LIN {X 0,Y 368.171,Z 278.475,A -85,B 0,C 180,E1 12084.523,E2 12084.523} C_VEL
LIN {X 0,Y 365.845,Z 275.09,A -85,B 0,C 180,E1 12082.497,E2 12082.497} C_VEL
LIN {X 0,Y 364.939,Z 273.089,A -85,B 0,C 180,E1 12081.371,E2 12081.371} C_VEL
LIN {X 0,Y 362.071,Z 268.956,A -85,B 0,C 180,E1 12077.685,E2 12077.685} C_VEL
LIN {X 0,Y 361.817,Z 267.734,A -85,B 0,C 180,E1 12076.208,E2 12076.208} C_VEL
LIN {X 0,Y 361.806,Z 267.661,A -85,B 0,C 180,E1 12072.125,E2 12072.125} C_VEL
LIN {X 0,Y 361.806,Z 267.652,A -85,B 0,C 180,E1 12067.943,E2 12067.943} C_VEL
LIN {X 0,Y 361.86,Z 268.035,A -85,B 0,C 180,E1 12064.438,E2 12064.438} C_VEL
LIN {X 0,Y 364.418,Z 272.635,A -85,B 0,C 180,E1 12060.316,E2 12060.316} C_VEL
LIN {X 0,Y 365.404,Z 274.131,A -85,B 0,C 180,E1 12059.217,E2 12059.217} C_VEL
LIN {X 0,Y 367.498,Z 277.914,A -85,B 0,C 180,E1 12057.038,E2 12057.038} C_VEL
LIN {X 0,Y 368.456,Z 279.19,A -85,B 0,C 180,E1 12056.267,E2 12056.267} C_VEL
LIN {X 0,Y 370.329,Z 282.88,A -85,B 0,C 180,E1 12054.579,E2 12054.579} C_VEL
LIN {X 0,Y 371.35,Z 284.531,A -85,B 0,C 180,E1 12053.819,E2 12053.819} C_VEL
LIN {X 0,Y 373.993,Z 289.456,A -85,B 0,C 180,E1 12051.856,E2 12051.856} C_VEL
LIN {X 0,Y 376.746,Z 294.987,A -85,B 0,C 180,E1 12049.913,E2 12049.913} C_VEL
LIN {X 0,Y 379.817,Z 300.91,A -85,B 0,C 180,E1 12048.075,E2 12048.075} C_VEL
LIN {X 0,Y 385.945,Z 309.361,A -85,B 0,C 180,E1 12046.293,E2 12046.293} C_VEL
LIN {X 0,Y 394.032,Z 321.193,A -85,B 0,C 180,E1 12044.158,E2 12044.158} C_VEL
LIN {X 0,Y 402.897,Z 335.236,A -85,B 0,C 180,E1 12042.042,E2 12042.042} C_VEL
LIN {X 0,Y 410.49,Z 348.634,A -85,B 0,C 180,E1 12040.362,E2 12040.362} C_VEL
LIN {X 0,Y 399.537,Z 571.468,A -85,B 0,C 180,E1 12035.877,E2 12035.877} C_VEL
LIN {X 0,Y 397.756,Z 592.269,A -85,B 0,C 180,E1 12035.206,E2 12035.206} C_VEL
LIN {X 0,Y 395.491,Z 611.619,A -85,B 0,C 180,E1 12034.346,E2 12034.346} C_VEL
LIN {X 0,Y 392.522,Z 632.048,A -85,B 0,C 180,E1 12033.159,E2 12033.159} C_VEL
LIN {X 0,Y 389.245,Z 650.935,A -85,B 0,C 180,E1 12031.774,E2 12031.774} C_VEL
LIN {X 0,Y 385.65,Z 668.995,A -85,B 0,C 180,E1 12030.148,E2 12030.148} C_VEL
LIN {X 0,Y 381.789,Z 686.588,A -85,B 0,C 180,E1 12028.209,E2 12028.209} C_VEL
LIN {X 0,Y 377.954,Z 702.615,A -85,B 0,C 180,E1 12026.071,E2 12026.071} C_VEL
LIN {X 0,Y 374.362,Z 717.031,A -85,B 0,C 180,E1 12023.766,E2 12023.766} C_VEL
LIN {X 0,Y 370.819,Z 731.031,A -85,B 0,C 180,E1 12021.081,E2 12021.081} C_VEL
LIN {X 0,Y 367.884,Z 742.762,A -85,B 0,C 180,E1 12018.369,E2 12018.369} C_VEL
LIN {X 0,Y 365.466,Z 752.896,A -85,B 0,C 180,E1 12015.546,E2 12015.546} C_VEL
LIN {X 0,Y 363.43,Z 762.078,A -85,B 0,C 180,E1 12012.381,E2 12012.381} C_VEL
LIN {X 0,Y 362.031,Z 769.268,A -85,B 0,C 180,E1 12009.233,E2 12009.233} C_VEL
LIN {X 0,Y 361.116,Z 774.969,A -85,B 0,C 180,E1 12005.945,E2 12005.945} C_VEL
LIN {X 0,Y 360.61,Z 779.064,A -85,B 0,C 180,E1 12002.542,E2 12002.542} C_VEL
LIN {X 0,Y 360.405,Z 781.321,A -85,B 0,C 180,E1 11999.411,E2 11999.411} C_VEL
LIN {X 0,Y 360.342,Z 782.079,A -85,B 0,C 180,E1 11996.336,E2 11996.336} C_VEL
LIN {X 0,Y 360.361,Z 781.41,A -85,B 0,C 180,E1 11993.205,E2 11993.205} C_VEL
LIN {X 0,Y 360.519,Z 779.191,A -85,B 0,C 180,E1 11989.925,E2 11989.925} C_VEL
LIN {X 0,Y 360.9,Z 775.517,A -85,B 0,C 180,E1 11986.747,E2 11986.747} C_VEL
LIN {X 0,Y 361.665,Z 769.902,A -85,B 0,C 180,E1 11983.43,E2 11983.43} C_VEL
LIN {X 0,Y 362.853,Z 762.904,A -85,B 0,C 180,E1 11980.32,E2 11980.32} C_VEL
LIN {X 0,Y 364.579,Z 754.204,A -85,B 0,C 180,E1 11977.249,E2 11977.249} C_VEL
LIN {X 0,Y 366.111,Z 747.184,A -85,B 0,C 180,E1 11975.17,E2 11975.17} C_VEL
LIN {X 0,Y 366.048,Z 743.524,A -85,B 0,C 180,E1 11974.098,E2 11974.098} C_VEL
LIN {X 0,Y 362.759,Z 733.509,A -85,B 0,C 180,E1 11971.203,E2 11971.203} C_VEL
LIN {X 0,Y 363.017,Z 729.697,A -85,B 0,C 180,E1 11970.335,E2 11970.335} C_VEL
LIN {X 0,Y 366.543,Z 715.603,A -85,B 0,C 180,E1 11967.657,E2 11967.657} C_VEL
LIN {X 0,Y 370.168,Z 700.835,A -85,B 0,C 180,E1 11965.319,E2 11965.319} C_VEL
LIN {X 0,Y 373.855,Z 685.185,A -85,B 0,C 180,E1 11963.244,E2 11963.244} C_VEL
LIN {X 0,Y 377.797,Z 666.968,A -85,B 0,C 180,E1 11961.249,E2 11961.249} C_VEL
LIN {X 0,Y 381.444,Z 648.231,A -85,B 0,C 180,E1 11959.582,E2 11959.582} C_VEL
LIN {X 0,Y 384.61,Z 629.426,A -85,B 0,C 180,E1 11958.226,E2 11958.226} C_VEL
LIN {X 0,Y 387.367,Z 609.919,A -85,B 0,C 180,E1 11957.108,E2 11957.108} C_VEL
LIN {X 0,Y 389.704,Z 589.326,A -85,B 0,C 180,E1 11956.212,E2 11956.212} C_VEL
LIN {X 0,Y 391.382,Z 568.754,A -85,B 0,C 180,E1 11955.569,E2 11955.569} C_VEL
LIN {X 0,Y 401.198,Z 349.516,A -85,B 0,C 180,E1 11951.239,E2 11951.239} C_VEL
LIN {X 0,Y 390.797,Z 331.837,A -85,B 0,C 180,E1 11949.151,E2 11949.151} C_VEL
LIN {X 0,Y 380.876,Z 316.345,A -85,B 0,C 180,E1 11947.024,E2 11947.024} C_VEL
LIN {X 0,Y 369.459,Z 299.547,A -85,B 0,C 180,E1 11944.31,E2 11944.31} C_VEL
LIN {X 0,Y 363.406,Z 287.193,A -85,B 0,C 180,E1 11941.032,E2 11941.032} C_VEL
LIN {X 0,Y 360.31,Z 281.531,A -85,B 0,C 180,E1 11939.34,E2 11939.34} C_VEL
LIN {X 0,Y 358.366,Z 277.681,A -85,B 0,C 180,E1 11938.178,E2 11938.178} C_VEL
LIN {X 0,Y 356.111,Z 273.295,A -85,B 0,C 180,E1 11936.789,E2 11936.789} C_VEL
LIN {X 0,Y 354.135,Z 269.94,A -85,B 0,C 180,E1 11935.623,E2 11935.623} C_VEL
LIN {X 0,Y 353.858,Z 268.676,A -85,B 0,C 180,E1 11935.1,E2 11935.1} C_VEL
LIN {X 0,Y 353.852,Z 268.637,A -85,B 0,C 180,E1 11930.944,E2 11930.944} C_VEL
LIN {X 0,Y 353.853,Z 268.639,A -85,B 0,C 180,E1 11926.801,E2 11926.801} C_VEL
LIN {X 0,Y 353.855,Z 268.648,A -85,B 0,C 180,E1 11922.696,E2 11922.696} C_VEL
LIN {X 0,Y 353.858,Z 268.656,A -85,B 0,C 180,E1 11918.433,E2 11918.433} C_VEL
LIN {X 0,Y 353.864,Z 268.647,A -85,B 0,C 180,E1 11914.122,E2 11914.122} C_VEL
LIN {X 0,Y 353.873,Z 268.628,A -85,B 0,C 180,E1 11909.818,E2 11909.818} C_VEL
LIN {X 0,Y 353.866,Z 268.625,A -85,B 0,C 180,E1 11905.612,E2 11905.612} C_VEL
LIN {X 0,Y 353.872,Z 268.643,A -85,B 0,C 180,E1 11901.374,E2 11901.374} C_VEL
LIN {X 0,Y 353.864,Z 268.654,A -85,B 0,C 180,E1 11897.087,E2 11897.087} C_VEL
LIN {X 0,Y 353.859,Z 268.629,A -85,B 0,C 180,E1 11892.894,E2 11892.894} C_VEL
LIN {X 0,Y 353.856,Z 268.625,A -85,B 0,C 180,E1 11888.775,E2 11888.775} C_VEL
LIN {X 0,Y 353.857,Z 268.649,A -85,B 0,C 180,E1 11884.699,E2 11884.699} C_VEL
LIN {X 0,Y 353.854,Z 268.656,A -85,B 0,C 180,E1 11880.484,E2 11880.484} C_VEL
LIN {X 0,Y 353.847,Z 268.636,A -85,B 0,C 180,E1 11876.272,E2 11876.272} C_VEL
LIN {X 0,Y 353.843,Z 268.629,A -85,B 0,C 180,E1 11872.04,E2 11872.04} C_VEL
LIN {X 0,Y 353.844,Z 268.63,A -85,B 0,C 180,E1 11867.864,E2 11867.864} C_VEL
LIN {X 0,Y 353.844,Z 268.637,A -85,B 0,C 180,E1 11863.754,E2 11863.754} C_VEL
LIN {X 0,Y 353.846,Z 268.64,A -85,B 0,C 180,E1 11859.661,E2 11859.661} C_VEL
LIN {X 0,Y 353.913,Z 268.942,A -85,B 0,C 180,E1 11856.655,E2 11856.655} C_VEL
LIN {X 0,Y 355.339,Z 272.39,A -85,B 0,C 180,E1 11855.566,E2 11855.566} C_VEL
LIN {X 0,Y 356.893,Z 274.427,A -85,B 0,C 180,E1 11854.795,E2 11854.795} C_VEL
LIN {X 0,Y 358.766,Z 278.091,A -85,B 0,C 180,E1 11853.696,E2 11853.696} C_VEL
LIN {X 0,Y 359.707,Z 279.455,A -85,B 0,C 180,E1 11853.236,E2 11853.236} C_VEL
LIN {X 0,Y 362.062,Z 283.638,A -85,B 0,C 180,E1 11851.999,E2 11851.999} C_VEL
LIN {X 0,Y 368.063,Z 295.125,A -85,B 0,C 180,E1 11848.925,E2 11848.925} C_VEL
LIN {X 0,Y 371.968,Z 302.135,A -85,B 0,C 180,E1 11847.227,E2 11847.227} C_VEL
LIN {X 0,Y 385.1,Z 320.964,A -85,B 0,C 180,E1 11844.208,E2 11844.208} C_VEL
LIN {X 0,Y 397.504,Z 340.13,A -85,B 0,C 180,E1 11841.612,E2 11841.612} C_VEL
LIN {X 0,Y 405.844,Z 354.423,A -85,B 0,C 180,E1 11839.974,E2 11839.974} C_VEL
LIN {X 0,Y 397.273,Z 565.921,A -85,B 0,C 180,E1 11835.942,E2 11835.942} C_VEL
LIN {X 0,Y 395.586,Z 604.161,A -85,B 0,C 180,E1 11835.173,E2 11835.173} C_VEL
LIN {X 0,Y 393.543,Z 625.831,A -85,B 0,C 180,E1 11834.533,E2 11834.533} C_VEL
LIN {X 0,Y 390.884,Z 646.572,A -85,B 0,C 180,E1 11833.678,E2 11833.678} C_VEL
LIN {X 0,Y 387.766,Z 666.981,A -85,B 0,C 180,E1 11832.585,E2 11832.585} C_VEL
LIN {X 0,Y 384.063,Z 687.555,A -85,B 0,C 180,E1 11831.195,E2 11831.195} C_VEL
LIN {X 0,Y 380.11,Z 706.817,A -85,B 0,C 180,E1 11829.581,E2 11829.581} C_VEL
LIN {X 0,Y 375.81,Z 726.104,A -85,B 0,C 180,E1 11827.63,E2 11827.63} C_VEL
LIN {X 0,Y 371.717,Z 743.57,A -85,B 0,C 180,E1 11825.519,E2 11825.519} C_VEL
LIN {X 0,Y 367.661,Z 760.077,A -85,B 0,C 180,E1 11823.133,E2 11823.133} C_VEL
LIN {X 0,Y 363.946,Z 775.21,A -85,B 0,C 180,E1 11820.545,E2 11820.545} C_VEL
LIN {X 0,Y 360.639,Z 789.096,A -85,B 0,C 180,E1 11817.758,E2 11817.758} C_VEL
LIN {X 0,Y 357.812,Z 801.747,A -85,B 0,C 180,E1 11814.745,E2 11814.745} C_VEL
LIN {X 0,Y 355.593,Z 812.75,A -85,B 0,C 180,E1 11811.612,E2 11811.612} C_VEL
LIN {X 0,Y 353.937,Z 822.534,A -85,B 0,C 180,E1 11808.273,E2 11808.273} C_VEL
LIN {X 0,Y 352.897,Z 830.469,A -85,B 0,C 180,E1 11804.939,E2 11804.939} C_VEL
LIN {X 0,Y 352.357,Z 836.632,A -85,B 0,C 180,E1 11801.621,E2 11801.621} C_VEL
LIN {X 0,Y 352.155,Z 841.286,A -85,B 0,C 180,E1 11798.324,E2 11798.324} C_VEL
LIN {X 0,Y 352.148,Z 844.279,A -85,B 0,C 180,E1 11795.048,E2 11795.048} C_VEL
LIN {X 0,Y 352.177,Z 845.844,A -85,B 0,C 180,E1 11791.788,E2 11791.788} C_VEL
LIN {X 0,Y 352.189,Z 845.904,A -85,B 0,C 180,E1 11788.86,E2 11788.86} C_VEL
LIN {X 0,Y 352.155,Z 844.641,A -85,B 0,C 180,E1 11785.602,E2 11785.602} C_VEL
LIN {X 0,Y 352.151,Z 841.936,A -85,B 0,C 180,E1 11782.494,E2 11782.494} C_VEL
LIN {X 0,Y 352.305,Z 837.422,A -85,B 0,C 180,E1 11779.037,E2 11779.037} C_VEL
LIN {X 0,Y 352.749,Z 831.577,A -85,B 0,C 180,E1 11775.789,E2 11775.789} C_VEL
LIN {X 0,Y 353.717,Z 823.505,A -85,B 0,C 180,E1 11772.291,E2 11772.291} C_VEL
LIN {X 0,Y 355.282,Z 813.801,A -85,B 0,C 180,E1 11768.884,E2 11768.884} C_VEL
LIN {X 0,Y 357.524,Z 802.262,A -85,B 0,C 180,E1 11765.548,E2 11765.548} C_VEL
LIN {X 0,Y 360.232,Z 789.837,A -85,B 0,C 180,E1 11762.563,E2 11762.563} C_VEL
LIN {X 0,Y 363.661,Z 775.346,A -85,B 0,C 180,E1 11759.608,E2 11759.608} C_VEL
LIN {X 0,Y 367.455,Z 759.895,A -85,B 0,C 180,E1 11756.939,E2 11756.939} C_VEL
LIN {X 0,Y 371.492,Z 743.408,A -85,B 0,C 180,E1 11754.547,E2 11754.547} C_VEL
LIN {X 0,Y 375.747,Z 725.523,A -85,B 0,C 180,E1 11752.359,E2 11752.359} C_VEL
LIN {X 0,Y 380.019,Z 706.741,A -85,B 0,C 180,E1 11750.436,E2 11750.436} C_VEL
LIN {X 0,Y 384.069,Z 687.407,A -85,B 0,C 180,E1 11748.796,E2 11748.796} C_VEL
LIN {X 0,Y 387.78,Z 667.348,A -85,B 0,C 180,E1 11747.42,E2 11747.42} C_VEL
LIN {X 0,Y 391.268,Z 645.478,A -85,B 0,C 180,E1 11746.229,E2 11746.229} C_VEL
LIN {X 0,Y 394.075,Z 624.25,A -85,B 0,C 180,E1 11745.354,E2 11745.354} C_VEL
LIN {X 0,Y 396.163,Z 602.513,A -85,B 0,C 180,E1 11744.713,E2 11744.713} C_VEL
LIN {X 0,Y 397.935,Z 563.509,A -85,B 0,C 180,E1 11743.924,E2 11743.924} C_VEL
LIN {X 0,Y 406.612,Z 362.247,A -85,B 0,C 180,E1 11740.032,E2 11740.032} C_VEL
LIN {X 0,Y 406.892,Z 353.823,A -85,B 0,C 180,E1 11739.848,E2 11739.848} C_VEL
LIN {X 0,Y 398.203,Z 338.538,A -85,B 0,C 180,E1 11737.897,E2 11737.897} C_VEL
LIN {X 0,Y 389.857,Z 325.331,A -85,B 0,C 180,E1 11735.86,E2 11735.86} C_VEL
LIN {X 0,Y 381.451,Z 313.134,A -85,B 0,C 180,E1 11733.579,E2 11733.579} C_VEL
LIN {X 0,Y 374.48,Z 303.819,A -85,B 0,C 180,E1 11731.466,E2 11731.466} C_VEL
LIN {X 0,Y 372.423,Z 300.702,A -85,B 0,C 180,E1 11730.671,E2 11730.671} C_VEL
LIN {X 0,Y 369.278,Z 294.916,A -85,B 0,C 180,E1 11728.637,E2 11728.637} C_VEL
LIN {X 0,Y 366.686,Z 290.179,A -85,B 0,C 180,E1 11726.739,E2 11726.739} C_VEL
LIN {X 0,Y 364.476,Z 286.447,A -85,B 0,C 180,E1 11724.991,E2 11724.991} C_VEL
LIN {X 0,Y 363.776,Z 285.103,A -85,B 0,C 180,E1 11724.349,E2 11724.349} C_VEL
LIN {X 0,Y 361.487,Z 281.641,A -85,B 0,C 180,E1 11722.269,E2 11722.269} C_VEL
LIN {X 0,Y 360.76,Z 279.896,A -85,B 0,C 180,E1 11721.29,E2 11721.29} C_VEL
LIN {X 0,Y 357.919,Z 275.754,A -85,B 0,C 180,E1 11717.561,E2 11717.561} C_VEL
LIN {X 0,Y 357.203,Z 274.236,A -85,B 0,C 180,E1 11715.922,E2 11715.922} C_VEL
LIN {X 0,Y 355.791,Z 272.948,A -85,B 0,C 180,E1 11711.182,E2 11711.182} C_VEL
LIN {X 0,Y 356.483,Z 273.641,A -85,B 0,C 180,E1 11706.825,E2 11706.825} C_VEL
LIN {X 0,Y 357.675,Z 274.972,A -85,B 0,C 180,E1 11704.33,E2 11704.33} C_VEL
LIN {X 0,Y 360.059,Z 279.305,A -85,B 0,C 180,E1 11700.479,E2 11700.479} C_VEL
LIN {X 0,Y 360.971,Z 280.593,A -85,B 0,C 180,E1 11699.471,E2 11699.471} C_VEL
LIN {X 0,Y 363.034,Z 284.512,A -85,B 0,C 180,E1 11697.16,E2 11697.16} C_VEL
LIN {X 0,Y 363.802,Z 285.478,A -85,B 0,C 180,E1 11696.535,E2 11696.535} C_VEL
LIN {X 0,Y 365.818,Z 289.463,A -85,B 0,C 180,E1 11694.669,E2 11694.669} C_VEL
LIN {X 0,Y 366.727,Z 291.216,A -85,B 0,C 180,E1 11693.898,E2 11693.898} C_VEL
LIN {X 0,Y 369.138,Z 295.706,A -85,B 0,C 180,E1 11692.061,E2 11692.061} C_VEL
LIN {X 0,Y 371.718,Z 300.754,A -85,B 0,C 180,E1 11690.284,E2 11690.284} C_VEL
LIN {X 0,Y 379.116,Z 310.838,A -85,B 0,C 180,E1 11687.86,E2 11687.86} C_VEL
LIN {X 0,Y 384.806,Z 318.805,A -85,B 0,C 180,E1 11686.209,E2 11686.209} C_VEL
LIN {X 0,Y 393.452,Z 331.999,A -85,B 0,C 180,E1 11683.921,E2 11683.921} C_VEL
LIN {X 0,Y 402.593,Z 347.489,A -85,B 0,C 180,E1 11681.728,E2 11681.728} C_VEL
LIN {X 0,Y 405.119,Z 352.351,A -85,B 0,C 180,E1 11681.15,E2 11681.15} C_VEL
LIN {X 0,Y 393.789,Z 571.901,A -85,B 0,C 180,E1 11676.678,E2 11676.678} C_VEL
LIN {X 0,Y 391.933,Z 592.665,A -85,B 0,C 180,E1 11676.003,E2 11676.003} C_VEL
LIN {X 0,Y 389.485,Z 612.63,A -85,B 0,C 180,E1 11675.103,E2 11675.103} C_VEL
LIN {X 0,Y 386.367,Z 633.083,A -85,B 0,C 180,E1 11673.896,E2 11673.896} C_VEL
LIN {X 0,Y 382.894,Z 652.166,A -85,B 0,C 180,E1 11672.472,E2 11672.472} C_VEL
LIN {X 0,Y 379.319,Z 669.352,A -85,B 0,C 180,E1 11670.906,E2 11670.906} C_VEL
LIN {X 0,Y 375.234,Z 687.046,A -85,B 0,C 180,E1 11668.933,E2 11668.933} C_VEL
LIN {X 0,Y 371.199,Z 703.146,A -85,B 0,C 180,E1 11666.76,E2 11666.76} C_VEL
LIN {X 0,Y 367.346,Z 717.828,A -85,B 0,C 180,E1 11664.378,E2 11664.378} C_VEL
LIN {X 0,Y 363.718,Z 731.354,A -85,B 0,C 180,E1 11661.743,E2 11661.743} C_VEL
LIN {X 0,Y 360.512,Z 743.426,A -85,B 0,C 180,E1 11658.908,E2 11658.908} C_VEL
LIN {X 0,Y 357.828,Z 753.961,A -85,B 0,C 180,E1 11655.901,E2 11655.901} C_VEL
LIN {X 0,Y 355.665,Z 763.142,A -85,B 0,C 180,E1 11652.651,E2 11652.651} C_VEL
LIN {X 0,Y 354.14,Z 770.471,A -85,B 0,C 180,E1 11649.325,E2 11649.325} C_VEL
LIN {X 0,Y 353.201,Z 775.872,A -85,B 0,C 180,E1 11646.075,E2 11646.075} C_VEL
LIN {X 0,Y 352.66,Z 779.898,A -85,B 0,C 180,E1 11642.596,E2 11642.596} C_VEL
LIN {X 0,Y 352.43,Z 782.154,A -85,B 0,C 180,E1 11639.209,E2 11639.209} C_VEL
LIN {X 0,Y 352.37,Z 782.827,A -85,B 0,C 180,E1 11635.913,E2 11635.913} C_VEL
LIN {X 0,Y 352.41,Z 781.93,A -85,B 0,C 180,E1 11632.699,E2 11632.699} C_VEL
LIN {X 0,Y 352.604,Z 779.492,A -85,B 0,C 180,E1 11629.378,E2 11629.378} C_VEL
LIN {X 0,Y 353.091,Z 775.301,A -85,B 0,C 180,E1 11625.944,E2 11625.944} C_VEL
LIN {X 0,Y 353.951,Z 769.762,A -85,B 0,C 180,E1 11622.73,E2 11622.73} C_VEL
LIN {X 0,Y 355.386,Z 762.171,A -85,B 0,C 180,E1 11619.393,E2 11619.393} C_VEL
LIN {X 0,Y 357.464,Z 752.599,A -85,B 0,C 180,E1 11616.103,E2 11616.103} C_VEL
LIN {X 0,Y 359.942,Z 742.108,A -85,B 0,C 180,E1 11613.186,E2 11613.186} C_VEL
LIN {X 0,Y 362.943,Z 729.991,A -85,B 0,C 180,E1 11610.397,E2 11610.397} C_VEL
LIN {X 0,Y 363.017,Z 729.697,A -85,B 0,C 180,E1 11610.335,E2 11610.335} C_VEL
LIN {X 0,Y 363.276,Z 725.23,A -85,B 0,C 180,E1 11609.334,E2 11609.334} C_VEL
LIN {X 0,Y 360.943,Z 713.902,A -85,B 0,C 180,E1 11606.727,E2 11606.727} C_VEL
LIN {X 0,Y 361.384,Z 708.797,A -85,B 0,C 180,E1 11605.802,E2 11605.802} C_VEL
LIN {X 0,Y 365.243,Z 693.476,A -85,B 0,C 180,E1 11603.554,E2 11603.554} C_VEL
LIN {X 0,Y 369.208,Z 676.766,A -85,B 0,C 180,E1 11601.514,E2 11601.514} C_VEL
LIN {X 0,Y 373.175,Z 658.233,A -85,B 0,C 180,E1 11599.66,E2 11599.66} C_VEL
LIN {X 0,Y 376.74,Z 639.384,A -85,B 0,C 180,E1 11598.132,E2 11598.132} C_VEL
LIN {X 0,Y 379.858,Z 620.033,A -85,B 0,C 180,E1 11596.874,E2 11596.874} C_VEL
LIN {X 0,Y 382.617,Z 598.881,A -85,B 0,C 180,E1 11595.808,E2 11595.808} C_VEL
LIN {X 0,Y 384.726,Z 577.543,A -85,B 0,C 180,E1 11595.029,E2 11595.029} C_VEL
LIN {X 0,Y 386.119,Z 555.392,A -85,B 0,C 180,E1 11594.487,E2 11594.487} C_VEL
LIN {X 0,Y 395.493,Z 352.855,A -85,B 0,C 180,E1 11590.469,E2 11590.469} C_VEL
LIN {X 0,Y 384.578,Z 334.275,A -85,B 0,C 180,E1 11588.194,E2 11588.194} C_VEL
LIN {X 0,Y 373.601,Z 317.34,A -85,B 0,C 180,E1 11585.723,E2 11585.723} C_VEL
LIN {X 0,Y 364.389,Z 304.199,A -85,B 0,C 180,E1 11583.486,E2 11583.486} C_VEL
LIN {X 0,Y 361.111,Z 299.359,A -85,B 0,C 180,E1 11582.55,E2 11582.55} C_VEL
LIN {X 0,Y 355.957,Z 288.76,A -85,B 0,C 180,E1 11579.576,E2 11579.576} C_VEL
LIN {X 0,Y 352.905,Z 283.238,A -85,B 0,C 180,E1 11577.818,E2 11577.818} C_VEL
LIN {X 0,Y 350.988,Z 279.336,A -85,B 0,C 180,E1 11576.577,E2 11576.577} C_VEL
LIN {X 0,Y 348.936,Z 275.745,A -85,B 0,C 180,E1 11575.32,E2 11575.32} C_VEL
LIN {X 0,Y 348.005,Z 274.092,A -85,B 0,C 180,E1 11574.728,E2 11574.728} C_VEL
LIN {X 0,Y 346.094,Z 270.562,A -85,B 0,C 180,E1 11573.427,E2 11573.427} C_VEL
LIN {X 0,Y 345.919,Z 269.661,A -85,B 0,C 180,E1 11572.838,E2 11572.838} C_VEL
LIN {X 0,Y 345.922,Z 269.637,A -85,B 0,C 180,E1 11568.558,E2 11568.558} C_VEL
LIN {X 0,Y 345.926,Z 269.633,A -85,B 0,C 180,E1 11564.211,E2 11564.211} C_VEL
LIN {X 0,Y 345.931,Z 269.621,A -85,B 0,C 180,E1 11559.913,E2 11559.913} C_VEL
LIN {X 0,Y 345.925,Z 269.613,A -85,B 0,C 180,E1 11555.692,E2 11555.692} C_VEL
LIN {X 0,Y 345.931,Z 269.615,A -85,B 0,C 180,E1 11551.503,E2 11551.503} C_VEL
LIN {X 0,Y 345.928,Z 269.637,A -85,B 0,C 180,E1 11547.171,E2 11547.171} C_VEL
LIN {X 0,Y 345.923,Z 269.641,A -85,B 0,C 180,E1 11542.965,E2 11542.965} C_VEL
LIN {X 0,Y 345.913,Z 269.616,A -85,B 0,C 180,E1 11538.712,E2 11538.712} C_VEL
LIN {X 0,Y 345.908,Z 269.612,A -85,B 0,C 180,E1 11534.468,E2 11534.468} C_VEL
LIN {X 0,Y 345.911,Z 269.634,A -85,B 0,C 180,E1 11530.154,E2 11530.154} C_VEL
LIN {X 0,Y 345.914,Z 269.647,A -85,B 0,C 180,E1 11525.971,E2 11525.971} C_VEL
LIN {X 0,Y 345.919,Z 269.622,A -85,B 0,C 180,E1 11521.655,E2 11521.655} C_VEL
LIN {X 0,Y 345.918,Z 269.613,A -85,B 0,C 180,E1 11517.514,E2 11517.514} C_VEL
LIN {X 0,Y 345.935,Z 269.616,A -85,B 0,C 180,E1 11513.193,E2 11513.193} C_VEL
LIN {X 0,Y 345.928,Z 269.628,A -85,B 0,C 180,E1 11509.001,E2 11509.001} C_VEL
LIN {X 0,Y 345.933,Z 269.637,A -85,B 0,C 180,E1 11504.75,E2 11504.75} C_VEL
LIN {X 0,Y 345.919,Z 269.638,A -85,B 0,C 180,E1 11500.409,E2 11500.409} C_VEL
LIN {X 0,Y 345.974,Z 269.9,A -85,B 0,C 180,E1 11498.822,E2 11498.822} C_VEL
LIN {X 0,Y 347.342,Z 273.305,A -85,B 0,C 180,E1 11497.667,E2 11497.667} C_VEL
LIN {X 0,Y 348.915,Z 275.084,A -85,B 0,C 180,E1 11496.883,E2 11496.883} C_VEL
LIN {X 0,Y 350.583,Z 278.721,A -85,B 0,C 180,E1 11495.751,E2 11495.751} C_VEL
LIN {X 0,Y 351.847,Z 280.308,A -85,B 0,C 180,E1 11495.128,E2 11495.128} C_VEL
LIN {X 0,Y 354.001,Z 284.439,A -85,B 0,C 180,E1 11493.856,E2 11493.856} C_VEL
LIN {X 0,Y 357.753,Z 291.307,A -85,B 0,C 180,E1 11491.814,E2 11491.814} C_VEL
LIN {X 0,Y 362.576,Z 300.412,A -85,B 0,C 180,E1 11489.324,E2 11489.324} C_VEL
LIN {X 0,Y 365.385,Z 304.531,A -85,B 0,C 180,E1 11488.488,E2 11488.488} C_VEL
LIN {X 0,Y 376.936,Z 320.677,A -85,B 0,C 180,E1 11485.689,E2 11485.689} C_VEL
LIN {X 0,Y 388.911,Z 339.001,A -85,B 0,C 180,E1 11483.038,E2 11483.038} C_VEL
LIN {X 0,Y 399.643,Z 356.661,A -85,B 0,C 180,E1 11480.845,E2 11480.845} C_VEL
LIN {X 0,Y 400.16,Z 358.051,A -85,B 0,C 180,E1 11480.73,E2 11480.73} C_VEL
LIN {X 0,Y 391.142,Z 571.042,A -85,B 0,C 180,E1 11476.627,E2 11476.627} C_VEL
LIN {X 0,Y 389.53,Z 604.571,A -85,B 0,C 180,E1 11475.933,E2 11475.933} C_VEL
LIN {X 0,Y 387.377,Z 626.504,A -85,B 0,C 180,E1 11475.275,E2 11475.275} C_VEL
LIN {X 0,Y 384.526,Z 647.648,A -85,B 0,C 180,E1 11474.381,E2 11474.381} C_VEL
LIN {X 0,Y 381.112,Z 668.76,A -85,B 0,C 180,E1 11473.212,E2 11473.212} C_VEL
LIN {X 0,Y 377.47,Z 688.165,A -85,B 0,C 180,E1 11471.872,E2 11471.872} C_VEL
LIN {X 0,Y 373.282,Z 707.629,A -85,B 0,C 180,E1 11470.203,E2 11470.203} C_VEL
LIN {X 0,Y 368.898,Z 726.345,A -85,B 0,C 180,E1 11468.264,E2 11468.264} C_VEL
LIN {X 0,Y 364.484,Z 744.244,A -85,B 0,C 180,E1 11466.042,E2 11466.042} C_VEL
LIN {X 0,Y 360.335,Z 760.447,A -85,B 0,C 180,E1 11463.649,E2 11463.649} C_VEL
LIN {X 0,Y 356.526,Z 775.178,A -85,B 0,C 180,E1 11461.063,E2 11461.063} C_VEL
LIN {X 0,Y 352.879,Z 789.692,A -85,B 0,C 180,E1 11458.055,E2 11458.055} C_VEL
LIN {X 0,Y 349.983,Z 802.091,A -85,B 0,C 180,E1 11455.01,E2 11455.01} C_VEL
LIN {X 0,Y 347.625,Z 813.216,A -85,B 0,C 180,E1 11451.714,E2 11451.714} C_VEL
LIN {X 0,Y 345.888,Z 823.044,A -85,B 0,C 180,E1 11448.19,E2 11448.19} C_VEL
LIN {X 0,Y 344.858,Z 830.757,A -85,B 0,C 180,E1 11444.78,E2 11444.78} C_VEL
LIN {X 0,Y 344.338,Z 836.699,A -85,B 0,C 180,E1 11441.386,E2 11441.386} C_VEL
LIN {X 0,Y 344.164,Z 841.257,A -85,B 0,C 180,E1 11437.831,E2 11437.831} C_VEL
LIN {X 0,Y 344.172,Z 843.917,A -85,B 0,C 180,E1 11434.664,E2 11434.664} C_VEL
LIN {X 0,Y 344.214,Z 845.199,A -85,B 0,C 180,E1 11431.33,E2 11431.33} C_VEL
LIN {X 0,Y 344.214,Z 845.106,A -85,B 0,C 180,E1 11428.334,E2 11428.334} C_VEL
LIN {X 0,Y 344.182,Z 843.549,A -85,B 0,C 180,E1 11424.999,E2 11424.999} C_VEL
LIN {X 0,Y 344.183,Z 840.681,A -85,B 0,C 180,E1 11421.815,E2 11421.815} C_VEL
LIN {X 0,Y 344.385,Z 835.855,A -85,B 0,C 180,E1 11418.272,E2 11418.272} C_VEL
LIN {X 0,Y 344.942,Z 829.639,A -85,B 0,C 180,E1 11414.851,E2 11414.851} C_VEL
LIN {X 0,Y 346.043,Z 821.52,A -85,B 0,C 180,E1 11411.394,E2 11411.394} C_VEL
LIN {X 0,Y 347.844,Z 811.38,A -85,B 0,C 180,E1 11407.878,E2 11407.878} C_VEL
LIN {X 0,Y 350.227,Z 800.163,A -85,B 0,C 180,E1 11404.643,E2 11404.643} C_VEL
LIN {X 0,Y 353.38,Z 786.828,A -85,B 0,C 180,E1 11401.432,E2 11401.432} C_VEL
LIN {X 0,Y 356.9,Z 772.756,A -85,B 0,C 180,E1 11398.594,E2 11398.594} C_VEL
LIN {X 0,Y 361.285,Z 755.881,A -85,B 0,C 180,E1 11395.722,E2 11395.722} C_VEL
LIN {X 0,Y 365.487,Z 739.624,A -85,B 0,C 180,E1 11393.387,E2 11393.387} C_VEL
LIN {X 0,Y 369.956,Z 721.639,A -85,B 0,C 180,E1 11391.23,E2 11391.23} C_VEL
LIN {X 0,Y 374.398,Z 702.656,A -85,B 0,C 180,E1 11389.335,E2 11389.335} C_VEL
LIN {X 0,Y 378.729,Z 682.354,A -85,B 0,C 180,E1 11387.665,E2 11387.665} C_VEL
LIN {X 0,Y 382.633,Z 661.929,A -85,B 0,C 180,E1 11386.312,E2 11386.312} C_VEL
LIN {X 0,Y 385.824,Z 641.882,A -85,B 0,C 180,E1 11385.272,E2 11385.272} C_VEL
LIN {X 0,Y 388.686,Z 620.024,A -85,B 0,C 180,E1 11384.412,E2 11384.412} C_VEL
LIN {X 0,Y 390.704,Z 598.338,A -85,B 0,C 180,E1 11383.799,E2 11383.799} C_VEL
LIN {X 0,Y 400.982,Z 371.603,A -85,B 0,C 180,E1 11379.349,E2 11379.349} C_VEL
LIN {X 0,Y 401.57,Z 357.268,A -85,B 0,C 180,E1 11379.046,E2 11379.046} C_VEL
LIN {X 0,Y 393.149,Z 342.514,A -85,B 0,C 180,E1 11377.067,E2 11377.067} C_VEL
LIN {X 0,Y 384.57,Z 328.75,A -85,B 0,C 180,E1 11374.844,E2 11374.844} C_VEL
LIN {X 0,Y 376.015,Z 316.302,A -85,B 0,C 180,E1 11372.354,E2 11372.354} C_VEL
LIN {X 0,Y 368.313,Z 306.134,A -85,B 0,C 180,E1 11369.789,E2 11369.789} C_VEL
LIN {X 0,Y 364.545,Z 301.13,A -85,B 0,C 180,E1 11368.328,E2 11368.328} C_VEL
LIN {X 0,Y 361.97,Z 296.448,A -85,B 0,C 180,E1 11366.407,E2 11366.407} C_VEL
LIN {X 0,Y 359.79,Z 292.186,A -85,B 0,C 180,E1 11364.462,E2 11364.462} C_VEL
LIN {X 0,Y 357.159,Z 288.205,A -85,B 0,C 180,E1 11362.033,E2 11362.033} C_VEL
LIN {X 0,Y 356.409,Z 286.551,A -85,B 0,C 180,E1 11361.045,E2 11361.045} C_VEL
LIN {X 0,Y 353.667,Z 282.15,A -85,B 0,C 180,E1 11357.1,E2 11357.1} C_VEL
LIN {X 0,Y 352.939,Z 280.965,A -85,B 0,C 180,E1 11355.445,E2 11355.445} C_VEL
LIN {X 0,Y 351.763,Z 279.859,A -85,B 0,C 180,E1 11351.146,E2 11351.146} C_VEL
LIN {X 0,Y 352.407,Z 280.524,A -85,B 0,C 180,E1 11346.845,E2 11346.845} C_VEL
LIN {X 0,Y 353.511,Z 281.84,A -85,B 0,C 180,E1 11344.381,E2 11344.381} C_VEL
LIN {X 0,Y 355.843,Z 286.109,A -85,B 0,C 180,E1 11340.484,E2 11340.484} C_VEL
LIN {X 0,Y 356.617,Z 287.448,A -85,B 0,C 180,E1 11339.519,E2 11339.519} C_VEL
LIN {X 0,Y 358.785,Z 291.326,A -85,B 0,C 180,E1 11337.126,E2 11337.126} C_VEL
LIN {X 0,Y 359.644,Z 293.306,A -85,B 0,C 180,E1 11336.164,E2 11336.164} C_VEL
LIN {X 0,Y 361.856,Z 297.08,A -85,B 0,C 180,E1 11334.293,E2 11334.293} C_VEL
LIN {X 0,Y 364.193,Z 301.205,A -85,B 0,C 180,E1 11332.588,E2 11332.588} C_VEL
LIN {X 0,Y 371.844,Z 311.501,A -85,B 0,C 180,E1 11329.752,E2 11329.752} C_VEL
LIN {X 0,Y 379.217,Z 321.892,A -85,B 0,C 180,E1 11327.403,E2 11327.403} C_VEL
LIN {X 0,Y 387.109,Z 333.881,A -85,B 0,C 180,E1 11325.167,E2 11325.167} C_VEL
LIN {X 0,Y 395.407,Z 347.595,A -85,B 0,C 180,E1 11323.039,E2 11323.039} C_VEL
LIN {X 0,Y 399.855,Z 355.851,A -85,B 0,C 180,E1 11321.964,E2 11321.964} C_VEL
LIN {X 0,Y 388.118,Z 572.484,A -85,B 0,C 180,E1 11317.501,E2 11317.501} C_VEL
LIN {X 0,Y 386.187,Z 593.234,A -85,B 0,C 180,E1 11316.819,E2 11316.819} C_VEL
LIN {X 0,Y 383.641,Z 613.206,A -85,B 0,C 180,E1 11315.911,E2 11315.911} C_VEL
LIN {X 0,Y 380.424,Z 633.425,A -85,B 0,C 180,E1 11314.708,E2 11314.708} C_VEL
LIN {X 0,Y 376.869,Z 652.182,A -85,B 0,C 180,E1 11313.3,E2 11313.3} C_VEL
LIN {X 0,Y 372.843,Z 670.616,A -85,B 0,C 180,E1 11311.596,E2 11311.596} C_VEL
LIN {X 0,Y 368.611,Z 688.152,A -85,B 0,C 180,E1 11309.609,E2 11309.609} C_VEL
LIN {X 0,Y 364.373,Z 704.205,A -85,B 0,C 180,E1 11307.399,E2 11307.399} C_VEL
LIN {X 0,Y 360.442,Z 718.377,A -85,B 0,C 180,E1 11305.058,E2 11305.058} C_VEL
LIN {X 0,Y 356.477,Z 732.395,A -85,B 0,C 180,E1 11302.277,E2 11302.277} C_VEL
LIN {X 0,Y 353.061,Z 744.514,A -85,B 0,C 180,E1 11299.359,E2 11299.359} C_VEL
LIN {X 0,Y 350.233,Z 754.931,A -85,B 0,C 180,E1 11296.304,E2 11296.304} C_VEL
LIN {X 0,Y 348.027,Z 763.683,A -85,B 0,C 180,E1 11293.14,E2 11293.14} C_VEL
LIN {X 0,Y 346.406,Z 770.837,A -85,B 0,C 180,E1 11289.849,E2 11289.849} C_VEL
LIN {X 0,Y 345.381,Z 776.211,A -85,B 0,C 180,E1 11286.611,E2 11286.611} C_VEL
LIN {X 0,Y 344.781,Z 780.216,A -85,B 0,C 180,E1 11283.238,E2 11283.238} C_VEL
LIN {X 0,Y 344.503,Z 782.7,A -85,B 0,C 180,E1 11279.801,E2 11279.801} C_VEL
LIN {X 0,Y 344.406,Z 783.5,A -85,B 0,C 180,E1 11276.558,E2 11276.558} C_VEL
LIN {X 0,Y 344.426,Z 782.903,A -85,B 0,C 180,E1 11273.255,E2 11273.255} C_VEL
LIN {X 0,Y 344.597,Z 780.864,A -85,B 0,C 180,E1 11269.939,E2 11269.939} C_VEL
LIN {X 0,Y 345.04,Z 777.128,A -85,B 0,C 180,E1 11266.5,E2 11266.5} C_VEL
LIN {X 0,Y 345.896,Z 771.639,A -85,B 0,C 180,E1 11263.067,E2 11263.067} C_VEL
LIN {X 0,Y 347.247,Z 764.666,A -85,B 0,C 180,E1 11259.783,E2 11259.783} C_VEL
LIN {X 0,Y 349.302,Z 755.552,A -85,B 0,C 180,E1 11256.411,E2 11256.411} C_VEL
LIN {X 0,Y 351.934,Z 744.943,A -85,B 0,C 180,E1 11253.259,E2 11253.259} C_VEL
LIN {X 0,Y 354.946,Z 733.428,A -85,B 0,C 180,E1 11250.441,E2 11250.441} C_VEL
LIN {X 0,Y 358.428,Z 720.249,A -85,B 0,C 180,E1 11247.764,E2 11247.764} C_VEL
LIN {X 0,Y 361.384,Z 708.797,A -85,B 0,C 180,E1 11245.802,E2 11245.802} C_VEL
LIN {X 0,Y 361.903,Z 703.596,A -85,B 0,C 180,E1 11244.891,E2 11244.891} C_VEL
LIN {X 0,Y 360.223,Z 690.498,A -85,B 0,C 180,E1 11242.481,E2 11242.481} C_VEL
LIN {X 0,Y 360.8,Z 684.716,A -85,B 0,C 180,E1 11241.666,E2 11241.666} C_VEL
LIN {X 0,Y 364.877,Z 667.388,A -85,B 0,C 180,E1 11239.742,E2 11239.742} C_VEL
LIN {X 0,Y 368.842,Z 648.511,A -85,B 0,C 180,E1 11238.033,E2 11238.033} C_VEL
LIN {X 0,Y 372.277,Z 629.481,A -85,B 0,C 180,E1 11236.647,E2 11236.647} C_VEL
LIN {X 0,Y 375.289,Z 609.52,A -85,B 0,C 180,E1 11235.498,E2 11235.498} C_VEL
LIN {X 0,Y 377.815,Z 588.282,A -85,B 0,C 180,E1 11234.578,E2 11234.578} C_VEL
LIN {X 0,Y 379.558,Z 567.452,A -85,B 0,C 180,E1 11233.94,E2 11233.94} C_VEL
LIN {X 0,Y 389.827,Z 356.154,A -85,B 0,C 180,E1 11229.677,E2 11229.677} C_VEL
LIN {X 0,Y 378.988,Z 337.794,A -85,B 0,C 180,E1 11227.332,E2 11227.332} C_VEL
LIN {X 0,Y 368.203,Z 321.085,A -85,B 0,C 180,E1 11224.811,E2 11224.811} C_VEL
LIN {X 0,Y 358.535,Z 307.221,A -85,B 0,C 180,E1 11222.342,E2 11222.342} C_VEL
LIN {X 0,Y 353.197,Z 299.841,A -85,B 0,C 180,E1 11220.865,E2 11220.865} C_VEL
LIN {X 0,Y 348.271,Z 289.95,A -85,B 0,C 180,E1 11217.874,E2 11217.874} C_VEL
LIN {X 0,Y 345.481,Z 284.886,A -85,B 0,C 180,E1 11216.157,E2 11216.157} C_VEL
LIN {X 0,Y 343.062,Z 280.304,A -85,B 0,C 180,E1 11214.553,E2 11214.553} C_VEL
LIN {X 0,Y 341.04,Z 276.601,A -85,B 0,C 180,E1 11213.163,E2 11213.163} C_VEL
LIN {X 0,Y 338.287,Z 272.026,A -85,B 0,C 180,E1 11211.284,E2 11211.284} C_VEL
LIN {X 0,Y 337.984,Z 270.653,A -85,B 0,C 180,E1 11210.65,E2 11210.65} C_VEL
LIN {X 0,Y 337.982,Z 270.609,A -85,B 0,C 180,E1 11206.429,E2 11206.429} C_VEL
LIN {X 0,Y 337.989,Z 270.61,A -85,B 0,C 180,E1 11202.057,E2 11202.057} C_VEL
LIN {X 0,Y 337.993,Z 270.62,A -85,B 0,C 180,E1 11197.757,E2 11197.757} C_VEL
LIN {X 0,Y 337.991,Z 270.633,A -85,B 0,C 180,E1 11193.381,E2 11193.381} C_VEL
LIN {X 0,Y 337.984,Z 270.618,A -85,B 0,C 180,E1 11189.021,E2 11189.021} C_VEL
LIN {X 0,Y 337.973,Z 270.603,A -85,B 0,C 180,E1 11184.744,E2 11184.744} C_VEL
LIN {X 0,Y 337.971,Z 270.605,A -85,B 0,C 180,E1 11180.43,E2 11180.43} C_VEL
LIN {X 0,Y 337.975,Z 270.628,A -85,B 0,C 180,E1 11176.144,E2 11176.144} C_VEL
LIN {X 0,Y 337.976,Z 270.624,A -85,B 0,C 180,E1 11171.95,E2 11171.95} C_VEL
LIN {X 0,Y 337.987,Z 270.602,A -85,B 0,C 180,E1 11167.649,E2 11167.649} C_VEL
LIN {X 0,Y 337.984,Z 270.603,A -85,B 0,C 180,E1 11163.39,E2 11163.39} C_VEL
LIN {X 0,Y 337.994,Z 270.617,A -85,B 0,C 180,E1 11159.151,E2 11159.151} C_VEL
LIN {X 0,Y 337.985,Z 270.632,A -85,B 0,C 180,E1 11154.737,E2 11154.737} C_VEL
LIN {X 0,Y 337.982,Z 270.622,A -85,B 0,C 180,E1 11150.635,E2 11150.635} C_VEL
LIN {X 0,Y 337.973,Z 270.616,A -85,B 0,C 180,E1 11146.309,E2 11146.309} C_VEL
LIN {X 0,Y 337.969,Z 270.615,A -85,B 0,C 180,E1 11142.08,E2 11142.08} C_VEL
LIN {X 0,Y 338.043,Z 271.002,A -85,B 0,C 180,E1 11141.165,E2 11141.165} C_VEL
LIN {X 0,Y 339.577,Z 274.524,A -85,B 0,C 180,E1 11139.848,E2 11139.848} C_VEL
LIN {X 0,Y 341.079,Z 276.1,A -85,B 0,C 180,E1 11139.044,E2 11139.044} C_VEL
LIN {X 0,Y 342.9,Z 280.008,A -85,B 0,C 180,E1 11137.723,E2 11137.723} C_VEL
LIN {X 0,Y 344.086,Z 281.546,A -85,B 0,C 180,E1 11137.083,E2 11137.083} C_VEL
LIN {X 0,Y 346.126,Z 285.438,A -85,B 0,C 180,E1 11135.782,E2 11135.782} C_VEL
LIN {X 0,Y 347.217,Z 287.377,A -85,B 0,C 180,E1 11135.137,E2 11135.137} C_VEL
LIN {X 0,Y 349.999,Z 292.433,A -85,B 0,C 180,E1 11133.534,E2 11133.534} C_VEL
LIN {X 0,Y 354.742,Z 301.048,A -85,B 0,C 180,E1 11131,E2 11131} C_VEL
LIN {X 0,Y 366.044,Z 316.682,A -85,B 0,C 180,E1 11127.953,E2 11127.953} C_VEL
LIN {X 0,Y 377.169,Z 332.913,A -85,B 0,C 180,E1 11125.275,E2 11125.275} C_VEL
LIN {X 0,Y 389.332,Z 352.124,A -85,B 0,C 180,E1 11122.6,E2 11122.6} C_VEL
LIN {X 0,Y 394.531,Z 361.269,A -85,B 0,C 180,E1 11121.511,E2 11121.511} C_VEL
LIN {X 0,Y 385.058,Z 576.371,A -85,B 0,C 180,E1 11117.33,E2 11117.33} C_VEL
LIN {X 0,Y 383.447,Z 606.098,A -85,B 0,C 180,E1 11116.688,E2 11116.688} C_VEL
LIN {X 0,Y 381.176,Z 627.82,A -85,B 0,C 180,E1 11116.014,E2 11116.014} C_VEL
LIN {X 0,Y 378.197,Z 648.865,A -85,B 0,C 180,E1 11115.098,E2 11115.098} C_VEL
LIN {X 0,Y 374.691,Z 669.424,A -85,B 0,C 180,E1 11113.929,E2 11113.929} C_VEL
LIN {X 0,Y 370.713,Z 689.517,A -85,B 0,C 180,E1 11112.5,E2 11112.5} C_VEL
LIN {X 0,Y 366.397,Z 708.825,A -85,B 0,C 180,E1 11110.809,E2 11110.809} C_VEL
LIN {X 0,Y 361.86,Z 727.266,A -85,B 0,C 180,E1 11108.843,E2 11108.843} C_VEL
LIN {X 0,Y 357.208,Z 745.189,A -85,B 0,C 180,E1 11106.549,E2 11106.549} C_VEL
LIN {X 0,Y 352.809,Z 761.586,A -85,B 0,C 180,E1 11104.05,E2 11104.05} C_VEL
LIN {X 0,Y 348.675,Z 776.863,A -85,B 0,C 180,E1 11101.265,E2 11101.265} C_VEL
LIN {X 0,Y 345.127,Z 790.275,A -85,B 0,C 180,E1 11098.365,E2 11098.365} C_VEL
LIN {X 0,Y 342.129,Z 802.469,A -85,B 0,C 180,E1 11095.255,E2 11095.255} C_VEL
LIN {X 0,Y 339.627,Z 813.826,A -85,B 0,C 180,E1 11091.772,E2 11091.772} C_VEL
LIN {X 0,Y 337.907,Z 823.113,A -85,B 0,C 180,E1 11088.277,E2 11088.277} C_VEL
LIN {X 0,Y 336.816,Z 831.011,A -85,B 0,C 180,E1 11084.588,E2 11084.588} C_VEL
LIN {X 0,Y 336.322,Z 836.763,A -85,B 0,C 180,E1 11081.14,E2 11081.14} C_VEL
LIN {X 0,Y 336.179,Z 840.855,A -85,B 0,C 180,E1 11077.69,E2 11077.69} C_VEL
LIN {X 0,Y 336.201,Z 843.516,A -85,B 0,C 180,E1 11074.262,E2 11074.262} C_VEL
LIN {X 0,Y 336.25,Z 844.529,A -85,B 0,C 180,E1 11071.02,E2 11071.02} C_VEL
LIN {X 0,Y 336.236,Z 844.257,A -85,B 0,C 180,E1 11067.659,E2 11067.659} C_VEL
LIN {X 0,Y 336.197,Z 842.449,A -85,B 0,C 180,E1 11064.366,E2 11064.366} C_VEL
LIN {X 0,Y 336.215,Z 839.116,A -85,B 0,C 180,E1 11060.87,E2 11060.87} C_VEL
LIN {X 0,Y 336.481,Z 834.289,A -85,B 0,C 180,E1 11057.47,E2 11057.47} C_VEL
LIN {X 0,Y 337.207,Z 827.43,A -85,B 0,C 180,E1 11053.814,E2 11053.814} C_VEL
LIN {X 0,Y 338.489,Z 819.188,A -85,B 0,C 180,E1 11050.32,E2 11050.32} C_VEL
LIN {X 0,Y 340.516,Z 808.853,A -85,B 0,C 180,E1 11046.791,E2 11046.791} C_VEL
LIN {X 0,Y 343.268,Z 796.929,A -85,B 0,C 180,E1 11043.409,E2 11043.409} C_VEL
LIN {X 0,Y 346.678,Z 783.606,A -85,B 0,C 180,E1 11040.242,E2 11040.242} C_VEL
LIN {X 0,Y 350.737,Z 768.612,A -85,B 0,C 180,E1 11037.243,E2 11037.243} C_VEL
LIN {X 0,Y 355.122,Z 752.437,A -85,B 0,C 180,E1 11034.548,E2 11034.548} C_VEL
LIN {X 0,Y 359.843,Z 734.967,A -85,B 0,C 180,E1 11032.104,E2 11032.104} C_VEL
LIN {X 0,Y 364.56,Z 716.684,A -85,B 0,C 180,E1 11029.961,E2 11029.961} C_VEL
LIN {X 0,Y 369.165,Z 697.655,A -85,B 0,C 180,E1 11028.114,E2 11028.114} C_VEL
LIN {X 0,Y 373.312,Z 678.581,A -85,B 0,C 180,E1 11026.606,E2 11026.606} C_VEL
LIN {X 0,Y 377.445,Z 657.052,A -85,B 0,C 180,E1 11025.231,E2 11025.231} C_VEL
LIN {X 0,Y 380.631,Z 637.629,A -85,B 0,C 180,E1 11024.252,E2 11024.252} C_VEL
LIN {X 0,Y 383.398,Z 616,A -85,B 0,C 180,E1 11023.446,E2 11023.446} C_VEL
LIN {X 0,Y 385.335,Z 593.528,A -85,B 0,C 180,E1 11022.852,E2 11022.852} C_VEL
LIN {X 0,Y 395.792,Z 373.825,A -85,B 0,C 180,E1 11018.499,E2 11018.499} C_VEL
LIN {X 0,Y 396.36,Z 360.835,A -85,B 0,C 180,E1 11018.22,E2 11018.22} C_VEL
LIN {X 0,Y 388.544,Z 347.018,A -85,B 0,C 180,E1 11016.291,E2 11016.291} C_VEL
LIN {X 0,Y 380.202,Z 333.534,A -85,B 0,C 180,E1 11014.021,E2 11014.021} C_VEL
LIN {X 0,Y 372.565,Z 322.332,A -85,B 0,C 180,E1 11011.692,E2 11011.692} C_VEL
LIN {X 0,Y 365.805,Z 313.176,A -85,B 0,C 180,E1 11009.338,E2 11009.338} C_VEL
LIN {X 0,Y 361.976,Z 308.109,A -85,B 0,C 180,E1 11007.829,E2 11007.829} C_VEL
LIN {X 0,Y 357.8,Z 302.983,A -85,B 0,C 180,E1 11006.024,E2 11006.024} C_VEL
LIN {X 0,Y 355.776,Z 299.995,A -85,B 0,C 180,E1 11004.756,E2 11004.756} C_VEL
LIN {X 0,Y 354.964,Z 298.293,A -85,B 0,C 180,E1 11003.931,E2 11003.931} C_VEL
LIN {X 0,Y 352.726,Z 294.394,A -85,B 0,C 180,E1 11001.598,E2 11001.598} C_VEL
LIN {X 0,Y 352.076,Z 293.208,A -85,B 0,C 180,E1 11000.794,E2 11000.794} C_VEL
LIN {X 0,Y 349.507,Z 288.759,A -85,B 0,C 180,E1 10996.795,E2 10996.795} C_VEL
LIN {X 0,Y 348.397,Z 287.419,A -85,B 0,C 180,E1 10994.29,E2 10994.29} C_VEL
LIN {X 0,Y 347.707,Z 286.76,A -85,B 0,C 180,E1 10989.769,E2 10989.769} C_VEL
LIN {X 0,Y 349.157,Z 288.221,A -85,B 0,C 180,E1 10984.93,E2 10984.93} C_VEL
LIN {X 0,Y 351.791,Z 293.062,A -85,B 0,C 180,E1 10980.327,E2 10980.327} C_VEL
LIN {X 0,Y 354.365,Z 297.956,A -85,B 0,C 180,E1 10977.247,E2 10977.247} C_VEL
LIN {X 0,Y 356.035,Z 301.373,A -85,B 0,C 180,E1 10975.653,E2 10975.653} C_VEL
LIN {X 0,Y 358.654,Z 304.559,A -85,B 0,C 180,E1 10974.421,E2 10974.421} C_VEL
LIN {X 0,Y 362.39,Z 309.279,A -85,B 0,C 180,E1 10972.79,E2 10972.79} C_VEL
LIN {X 0,Y 367.762,Z 316.517,A -85,B 0,C 180,E1 10970.726,E2 10970.726} C_VEL
LIN {X 0,Y 375.248,Z 326.994,A -85,B 0,C 180,E1 10968.201,E2 10968.201} C_VEL
LIN {X 0,Y 383.644,Z 340.117,A -85,B 0,C 180,E1 10965.705,E2 10965.705} C_VEL
LIN {X 0,Y 391.693,Z 353.724,A -85,B 0,C 180,E1 10963.561,E2 10963.561} C_VEL
LIN {X 0,Y 394.687,Z 359.515,A -85,B 0,C 180,E1 10962.8,E2 10962.8} C_VEL
LIN {X 0,Y 382.572,Z 572.946,A -85,B 0,C 180,E1 10958.356,E2 10958.356} C_VEL
LIN {X 0,Y 380.561,Z 593.661,A -85,B 0,C 180,E1 10957.668,E2 10957.668} C_VEL
LIN {X 0,Y 377.888,Z 613.759,A -85,B 0,C 180,E1 10956.747,E2 10956.747} C_VEL
LIN {X 0,Y 374.562,Z 633.8,A -85,B 0,C 180,E1 10955.545,E2 10955.545} C_VEL
LIN {X 0,Y 370.796,Z 652.883,A -85,B 0,C 180,E1 10954.1,E2 10954.1} C_VEL
LIN {X 0,Y 366.665,Z 671.024,A -85,B 0,C 180,E1 10952.407,E2 10952.407} C_VEL
LIN {X 0,Y 362.204,Z 688.615,A -85,B 0,C 180,E1 10950.39,E2 10950.39} C_VEL
LIN {X 0,Y 357.688,Z 704.966,A -85,B 0,C 180,E1 10948.11,E2 10948.11} C_VEL
LIN {X 0,Y 353.479,Z 719.379,A -85,B 0,C 180,E1 10945.688,E2 10945.688} C_VEL
LIN {X 0,Y 349.45,Z 732.841,A -85,B 0,C 180,E1 10942.968,E2 10942.968} C_VEL
LIN {X 0,Y 345.835,Z 744.951,A -85,B 0,C 180,E1 10940.011,E2 10940.011} C_VEL
LIN {X 0,Y 342.882,Z 755.194,A -85,B 0,C 180,E1 10936.975,E2 10936.975} C_VEL
LIN {X 0,Y 340.417,Z 764.226,A -85,B 0,C 180,E1 10933.65,E2 10933.65} C_VEL
LIN {X 0,Y 338.657,Z 771.417,A -85,B 0,C 180,E1 10930.286,E2 10930.286} C_VEL
LIN {X 0,Y 337.477,Z 777.125,A -85,B 0,C 180,E1 10926.762,E2 10926.762} C_VEL
LIN {X 0,Y 336.81,Z 781.225,A -85,B 0,C 180,E1 10923.11,E2 10923.11} C_VEL
LIN {X 0,Y 336.533,Z 783.484,A -85,B 0,C 180,E1 10919.748,E2 10919.748} C_VEL
LIN {X 0,Y 336.438,Z 784.23,A -85,B 0,C 180,E1 10916.475,E2 10916.475} C_VEL
LIN {X 0,Y 336.464,Z 783.569,A -85,B 0,C 180,E1 10913.097,E2 10913.097} C_VEL
LIN {X 0,Y 336.657,Z 781.474,A -85,B 0,C 180,E1 10909.705,E2 10909.705} C_VEL
LIN {X 0,Y 337.148,Z 777.706,A -85,B 0,C 180,E1 10906.188,E2 10906.188} C_VEL
LIN {X 0,Y 338.098,Z 772.103,A -85,B 0,C 180,E1 10902.643,E2 10902.643} C_VEL
LIN {X 0,Y 339.545,Z 765.138,A -85,B 0,C 180,E1 10899.322,E2 10899.322} C_VEL
LIN {X 0,Y 341.743,Z 756.002,A -85,B 0,C 180,E1 10895.892,E2 10895.892} C_VEL
LIN {X 0,Y 344.562,Z 745.289,A -85,B 0,C 180,E1 10892.663,E2 10892.663} C_VEL
LIN {X 0,Y 347.705,Z 733.909,A -85,B 0,C 180,E1 10889.837,E2 10889.837} C_VEL
LIN {X 0,Y 351.447,Z 720.462,A -85,B 0,C 180,E1 10887.066,E2 10887.066} C_VEL
LIN {X 0,Y 355.597,Z 705.103,A -85,B 0,C 180,E1 10884.459,E2 10884.459} C_VEL
LIN {X 0,Y 359.649,Z 689.384,A -85,B 0,C 180,E1 10882.253,E2 10882.253} C_VEL
LIN {X 0,Y 360.8,Z 684.716,A -85,B 0,C 180,E1 10881.666,E2 10881.666} C_VEL
LIN {X 0,Y 361.406,Z 678.881,A -85,B 0,C 180,E1 10880.873,E2 10880.873} C_VEL
LIN {X 0,Y 360.108,Z 664.104,A -85,B 0,C 180,E1 10878.7,E2 10878.7} C_VEL
LIN {X 0,Y 360.725,Z 657.744,A -85,B 0,C 180,E1 10878.005,E2 10878.005} C_VEL
LIN {X 0,Y 364.615,Z 638.553,A -85,B 0,C 180,E1 10876.442,E2 10876.442} C_VEL
LIN {X 0,Y 367.863,Z 619.401,A -85,B 0,C 180,E1 10875.199,E2 10875.199} C_VEL
LIN {X 0,Y 370.722,Z 598.74,A -85,B 0,C 180,E1 10874.159,E2 10874.159} C_VEL
LIN {X 0,Y 372.984,Z 577.013,A -85,B 0,C 180,E1 10873.368,E2 10873.368} C_VEL
LIN {X 0,Y 374.547,Z 552.577,A -85,B 0,C 180,E1 10872.78,E2 10872.78} C_VEL
LIN {X 0,Y 384.192,Z 359.457,A -85,B 0,C 180,E1 10868.856,E2 10868.856} C_VEL
LIN {X 0,Y 372.953,Z 340.401,A -85,B 0,C 180,E1 10866.324,E2 10866.324} C_VEL
LIN {X 0,Y 361.872,Z 323.393,A -85,B 0,C 180,E1 10863.611,E2 10863.611} C_VEL
LIN {X 0,Y 351.945,Z 309.416,A -85,B 0,C 180,E1 10860.95,E2 10860.95} C_VEL
LIN {X 0,Y 344.841,Z 299.585,A -85,B 0,C 180,E1 10858.794,E2 10858.794} C_VEL
LIN {X 0,Y 340.707,Z 291.351,A -85,B 0,C 180,E1 10856.114,E2 10856.114} C_VEL
LIN {X 0,Y 337.799,Z 286.109,A -85,B 0,C 180,E1 10854.192,E2 10854.192} C_VEL
LIN {X 0,Y 335.382,Z 281.57,A -85,B 0,C 180,E1 10852.464,E2 10852.464} C_VEL
LIN {X 0,Y 333.29,Z 277.966,A -85,B 0,C 180,E1 10850.953,E2 10850.953} C_VEL
LIN {X 0,Y 332.51,Z 276.442,A -85,B 0,C 180,E1 10850.332,E2 10850.332} C_VEL
LIN {X 0,Y 330.346,Z 273.018,A -85,B 0,C 180,E1 10848.717,E2 10848.717} C_VEL
LIN {X 0,Y 330.059,Z 271.656,A -85,B 0,C 180,E1 10847.976,E2 10847.976} C_VEL
LIN {X 0,Y 330.052,Z 271.621,A -85,B 0,C 180,E1 10843.616,E2 10843.616} C_VEL
LIN {X 0,Y 330.048,Z 271.608,A -85,B 0,C 180,E1 10839.28,E2 10839.28} C_VEL
LIN {X 0,Y 330.035,Z 271.598,A -85,B 0,C 180,E1 10834.818,E2 10834.818} C_VEL
LIN {X 0,Y 330.037,Z 271.589,A -85,B 0,C 180,E1 10830.391,E2 10830.391} C_VEL
LIN {X 0,Y 330.038,Z 271.596,A -85,B 0,C 180,E1 10826.249,E2 10826.249} C_VEL
LIN {X 0,Y 330.054,Z 271.617,A -85,B 0,C 180,E1 10821.875,E2 10821.875} C_VEL
LIN {X 0,Y 330.052,Z 271.614,A -85,B 0,C 180,E1 10817.404,E2 10817.404} C_VEL
LIN {X 0,Y 330.049,Z 271.588,A -85,B 0,C 180,E1 10813.131,E2 10813.131} C_VEL
LIN {X 0,Y 330.043,Z 271.589,A -85,B 0,C 180,E1 10808.886,E2 10808.886} C_VEL
LIN {X 0,Y 330.035,Z 271.608,A -85,B 0,C 180,E1 10804.516,E2 10804.516} C_VEL
LIN {X 0,Y 330.031,Z 271.625,A -85,B 0,C 180,E1 10800.172,E2 10800.172} C_VEL
LIN {X 0,Y 330.032,Z 271.607,A -85,B 0,C 180,E1 10795.829,E2 10795.829} C_VEL
LIN {X 0,Y 330.043,Z 271.596,A -85,B 0,C 180,E1 10791.462,E2 10791.462} C_VEL
LIN {X 0,Y 330.05,Z 271.593,A -85,B 0,C 180,E1 10787.044,E2 10787.044} C_VEL
LIN {X 0,Y 330.061,Z 271.846,A -85,B 0,C 180,E1 10783.907,E2 10783.907} C_VEL
LIN {X 0,Y 331.765,Z 275.657,A -85,B 0,C 180,E1 10782.277,E2 10782.277} C_VEL
LIN {X 0,Y 333.342,Z 277.668,A -85,B 0,C 180,E1 10781.279,E2 10781.279} C_VEL
LIN {X 0,Y 335.135,Z 281.178,A -85,B 0,C 180,E1 10779.933,E2 10779.933} C_VEL
LIN {X 0,Y 336.291,Z 282.505,A -85,B 0,C 180,E1 10779.278,E2 10779.278} C_VEL
LIN {X 0,Y 338.133,Z 286.303,A -85,B 0,C 180,E1 10777.941,E2 10777.941} C_VEL
LIN {X 0,Y 339.271,Z 287.987,A -85,B 0,C 180,E1 10777.279,E2 10777.279} C_VEL
LIN {X 0,Y 342.405,Z 293.782,A -85,B 0,C 180,E1 10775.317,E2 10775.317} C_VEL
LIN {X 0,Y 345.154,Z 298.846,A -85,B 0,C 180,E1 10773.69,E2 10773.69} C_VEL
LIN {X 0,Y 347.398,Z 302.341,A -85,B 0,C 180,E1 10772.672,E2 10772.672} C_VEL
LIN {X 0,Y 358.715,Z 317.727,A -85,B 0,C 180,E1 10769.469,E2 10769.469} C_VEL
LIN {X 0,Y 369.563,Z 333.221,A -85,B 0,C 180,E1 10766.715,E2 10766.715} C_VEL
LIN {X 0,Y 381.078,Z 351.319,A -85,B 0,C 180,E1 10764.027,E2 10764.027} C_VEL
LIN {X 0,Y 388.975,Z 364.583,A -85,B 0,C 180,E1 10762.313,E2 10762.313} C_VEL
LIN {X 0,Y 379.082,Z 580.071,A -85,B 0,C 180,E1 10758.083,E2 10758.083} C_VEL
LIN {X 0,Y 377.469,Z 607.028,A -85,B 0,C 180,E1 10757.48,E2 10757.48} C_VEL
LIN {X 0,Y 375.065,Z 628.711,A -85,B 0,C 180,E1 10756.787,E2 10756.787} C_VEL
LIN {X 0,Y 371.987,Z 649.679,A -85,B 0,C 180,E1 10755.859,E2 10755.859} C_VEL
LIN {X 0,Y 368.3,Z 670.249,A -85,B 0,C 180,E1 10754.66,E2 10754.66} C_VEL
LIN {X 0,Y 364.001,Z 690.862,A -85,B 0,C 180,E1 10753.152,E2 10753.152} C_VEL
LIN {X 0,Y 359.547,Z 709.939,A -85,B 0,C 180,E1 10751.438,E2 10751.438} C_VEL
LIN {X 0,Y 354.919,Z 727.874,A -85,B 0,C 180,E1 10749.474,E2 10749.474} C_VEL
LIN {X 0,Y 350.172,Z 745.325,A -85,B 0,C 180,E1 10747.189,E2 10747.189} C_VEL
LIN {X 0,Y 345.593,Z 761.639,A -85,B 0,C 180,E1 10744.645,E2 10744.645} C_VEL
LIN {X 0,Y 341.293,Z 776.787,A -85,B 0,C 180,E1 10741.823,E2 10741.823} C_VEL
LIN {X 0,Y 337.578,Z 790.105,A -85,B 0,C 180,E1 10738.865,E2 10738.865} C_VEL
LIN {X 0,Y 334.28,Z 802.821,A -85,B 0,C 180,E1 10735.511,E2 10735.511} C_VEL
LIN {X 0,Y 331.804,Z 813.547,A -85,B 0,C 180,E1 10732.126,E2 10732.126} C_VEL
LIN {X 0,Y 329.967,Z 822.923,A -85,B 0,C 180,E1 10728.476,E2 10728.476} C_VEL
LIN {X 0,Y 328.854,Z 830.533,A -85,B 0,C 180,E1 10724.791,E2 10724.791} C_VEL
LIN {X 0,Y 328.338,Z 836.274,A -85,B 0,C 180,E1 10721.236,E2 10721.236} C_VEL
LIN {X 0,Y 328.198,Z 840.295,A -85,B 0,C 180,E1 10717.702,E2 10717.702} C_VEL
LIN {X 0,Y 328.23,Z 842.871,A -85,B 0,C 180,E1 10714.191,E2 10714.191} C_VEL
LIN {X 0,Y 328.282,Z 843.813,A -85,B 0,C 180,E1 10711.045,E2 10711.045} C_VEL
LIN {X 0,Y 328.267,Z 843.582,A -85,B 0,C 180,E1 10707.729,E2 10707.729} C_VEL
LIN {X 0,Y 328.221,Z 841.855,A -85,B 0,C 180,E1 10704.404,E2 10704.404} C_VEL
LIN {X 0,Y 328.221,Z 838.866,A -85,B 0,C 180,E1 10701.061,E2 10701.061} C_VEL
LIN {X 0,Y 328.479,Z 834.099,A -85,B 0,C 180,E1 10697.517,E2 10697.517} C_VEL
LIN {X 0,Y 329.163,Z 827.81,A -85,B 0,C 180,E1 10693.952,E2 10693.952} C_VEL
LIN {X 0,Y 330.444,Z 819.739,A -85,B 0,C 180,E1 10690.373,E2 10690.373} C_VEL
LIN {X 0,Y 332.471,Z 809.833,A -85,B 0,C 180,E1 10686.797,E2 10686.797} C_VEL
LIN {X 0,Y 335.197,Z 798.593,A -85,B 0,C 180,E1 10683.419,E2 10683.419} C_VEL
LIN {X 0,Y 338.774,Z 785.254,A -85,B 0,C 180,E1 10680.079,E2 10680.079} C_VEL
LIN {X 0,Y 342.726,Z 771.169,A -85,B 0,C 180,E1 10677.135,E2 10677.135} C_VEL
LIN {X 0,Y 347.466,Z 754.73,A -85,B 0,C 180,E1 10674.241,E2 10674.241} C_VEL
LIN {X 0,Y 352.272,Z 738.009,A -85,B 0,C 180,E1 10671.773,E2 10671.773} C_VEL
LIN {X 0,Y 357.057,Z 720.458,A -85,B 0,C 180,E1 10669.613,E2 10669.613} C_VEL
LIN {X 0,Y 361.824,Z 701.854,A -85,B 0,C 180,E1 10667.708,E2 10667.708} C_VEL
LIN {X 0,Y 366.507,Z 681.895,A -85,B 0,C 180,E1 10666.027,E2 10666.027} C_VEL
LIN {X 0,Y 370.704,Z 661.758,A -85,B 0,C 180,E1 10664.661,E2 10664.661} C_VEL
LIN {X 0,Y 374.178,Z 641.773,A -85,B 0,C 180,E1 10663.6,E2 10663.6} C_VEL
LIN {X 0,Y 377.326,Z 619.782,A -85,B 0,C 180,E1 10662.713,E2 10662.713} C_VEL
LIN {X 0,Y 379.549,Z 597.988,A -85,B 0,C 180,E1 10662.081,E2 10662.081} C_VEL
LIN {X 0,Y 390.932,Z 372.009,A -85,B 0,C 180,E1 10657.544,E2 10657.544} C_VEL
LIN {X 0,Y 391.215,Z 364.339,A -85,B 0,C 180,E1 10657.364,E2 10657.364} C_VEL
LIN {X 0,Y 382.702,Z 349.256,A -85,B 0,C 180,E1 10655.131,E2 10655.131} C_VEL
LIN {X 0,Y 375.058,Z 337.043,A -85,B 0,C 180,E1 10652.901,E2 10652.901} C_VEL
LIN {X 0,Y 367.471,Z 325.775,A -85,B 0,C 180,E1 10650.396,E2 10650.396} C_VEL
LIN {X 0,Y 362.571,Z 319.268,A -85,B 0,C 180,E1 10648.586,E2 10648.586} C_VEL
LIN {X 0,Y 359.712,Z 315.291,A -85,B 0,C 180,E1 10647.39,E2 10647.39} C_VEL
LIN {X 0,Y 355.489,Z 310.006,A -85,B 0,C 180,E1 10645.49,E2 10645.49} C_VEL
LIN {X 0,Y 351.948,Z 305.497,A -85,B 0,C 180,E1 10643.615,E2 10643.615} C_VEL
LIN {X 0,Y 348.545,Z 301.211,A -85,B 0,C 180,E1 10641.455,E2 10641.455} C_VEL
LIN {X 0,Y 347.921,Z 300.023,A -85,B 0,C 180,E1 10640.701,E2 10640.701} C_VEL
LIN {X 0,Y 345.391,Z 295.538,A -85,B 0,C 180,E1 10636.621,E2 10636.621} C_VEL
LIN {X 0,Y 344.181,Z 294.167,A -85,B 0,C 180,E1 10633.782,E2 10633.782} C_VEL
LIN {X 0,Y 343.681,Z 293.711,A -85,B 0,C 180,E1 10629.209,E2 10629.209} C_VEL
LIN {X 0,Y 345.091,Z 295.207,A -85,B 0,C 180,E1 10624.821,E2 10624.821} C_VEL
LIN {X 0,Y 347.295,Z 299.598,A -85,B 0,C 180,E1 10620.661,E2 10620.661} C_VEL
LIN {X 0,Y 348.073,Z 301.129,A -85,B 0,C 180,E1 10619.672,E2 10619.672} C_VEL
LIN {X 0,Y 352.496,Z 306.652,A -85,B 0,C 180,E1 10616.912,E2 10616.912} C_VEL
LIN {X 0,Y 356.575,Z 311.902,A -85,B 0,C 180,E1 10614.813,E2 10614.813} C_VEL
LIN {X 0,Y 360.193,Z 316.598,A -85,B 0,C 180,E1 10613.186,E2 10613.186} C_VEL
LIN {X 0,Y 365.394,Z 323.762,A -85,B 0,C 180,E1 10611.115,E2 10611.115} C_VEL
LIN {X 0,Y 372.414,Z 333.904,A -85,B 0,C 180,E1 10608.66,E2 10608.66} C_VEL
LIN {X 0,Y 380.272,Z 346.453,A -85,B 0,C 180,E1 10606.236,E2 10606.236} C_VEL
LIN {X 0,Y 387.964,Z 359.743,A -85,B 0,C 180,E1 10604.109,E2 10604.109} C_VEL
LIN {X 0,Y 389.631,Z 363.18,A -85,B 0,C 180,E1 10603.66,E2 10603.66} C_VEL
LIN {X 0,Y 377.12,Z 573.429,A -85,B 0,C 180,E1 10599.236,E2 10599.236} C_VEL
LIN {X 0,Y 375.026,Z 594.179,A -85,B 0,C 180,E1 10598.542,E2 10598.542} C_VEL
LIN {X 0,Y 372.243,Z 614.342,A -85,B 0,C 180,E1 10597.611,E2 10597.611} C_VEL
LIN {X 0,Y 368.792,Z 634.304,A -85,B 0,C 180,E1 10596.404,E2 10596.404} C_VEL
LIN {X 0,Y 364.941,Z 653.034,A -85,B 0,C 180,E1 10594.976,E2 10594.976} C_VEL
LIN {X 0,Y 360.567,Z 671.454,A -85,B 0,C 180,E1 10593.244,E2 10593.244} C_VEL
LIN {X 0,Y 355.927,Z 688.945,A -85,B 0,C 180,E1 10591.22,E2 10591.22} C_VEL
LIN {X 0,Y 351.355,Z 704.752,A -85,B 0,C 180,E1 10589,E2 10589} C_VEL
LIN {X 0,Y 347.008,Z 718.934,A -85,B 0,C 180,E1 10586.612,E2 10586.612} C_VEL
LIN {X 0,Y 342.793,Z 732.382,A -85,B 0,C 180,E1 10583.898,E2 10583.898} C_VEL
LIN {X 0,Y 339.06,Z 744.207,A -85,B 0,C 180,E1 10581.028,E2 10581.028} C_VEL
LIN {X 0,Y 335.575,Z 755.439,A -85,B 0,C 180,E1 10577.675,E2 10577.675} C_VEL
LIN {X 0,Y 332.965,Z 764.283,A -85,B 0,C 180,E1 10574.385,E2 10574.385} C_VEL
LIN {X 0,Y 331.025,Z 771.607,A -85,B 0,C 180,E1 10570.955,E2 10570.955} C_VEL
LIN {X 0,Y 329.69,Z 777.471,A -85,B 0,C 180,E1 10567.342,E2 10567.342} C_VEL
LIN {X 0,Y 328.948,Z 781.552,A -85,B 0,C 180,E1 10563.798,E2 10563.798} C_VEL
LIN {X 0,Y 328.597,Z 784.058,A -85,B 0,C 180,E1 10560.218,E2 10560.218} C_VEL
LIN {X 0,Y 328.471,Z 784.927,A -85,B 0,C 180,E1 10556.778,E2 10556.778} C_VEL
LIN {X 0,Y 328.496,Z 784.315,A -85,B 0,C 180,E1 10553.121,E2 10553.121} C_VEL
LIN {X 0,Y 328.694,Z 782.333,A -85,B 0,C 180,E1 10549.736,E2 10549.736} C_VEL
LIN {X 0,Y 329.184,Z 778.714,A -85,B 0,C 180,E1 10546.228,E2 10546.228} C_VEL
LIN {X 0,Y 330.104,Z 773.532,A -85,B 0,C 180,E1 10542.769,E2 10542.769} C_VEL
LIN {X 0,Y 331.67,Z 766.412,A -85,B 0,C 180,E1 10539.196,E2 10539.196} C_VEL
LIN {X 0,Y 333.834,Z 757.895,A -85,B 0,C 180,E1 10535.846,E2 10535.846} C_VEL
LIN {X 0,Y 336.549,Z 748.118,A -85,B 0,C 180,E1 10532.726,E2 10532.726} C_VEL
LIN {X 0,Y 340.146,Z 735.659,A -85,B 0,C 180,E1 10529.497,E2 10529.497} C_VEL
LIN {X 0,Y 344.01,Z 722.322,A -85,B 0,C 180,E1 10526.669,E2 10526.669} C_VEL
LIN {X 0,Y 348.067,Z 708.021,A -85,B 0,C 180,E1 10524.149,E2 10524.149} C_VEL
LIN {X 0,Y 352.346,Z 692.33,A -85,B 0,C 180,E1 10521.845,E2 10521.845} C_VEL
LIN {X 0,Y 356.549,Z 675.763,A -85,B 0,C 180,E1 10519.82,E2 10519.82} C_VEL
LIN {X 0,Y 360.725,Z 657.744,A -85,B 0,C 180,E1 10518.005,E2 10518.005} C_VEL
LIN {X 0,Y 361.346,Z 651.233,A -85,B 0,C 180,E1 10517.338,E2 10517.338} C_VEL
LIN {X 0,Y 359.957,Z 635.054,A -85,B 0,C 180,E1 10515.451,E2 10515.451} C_VEL
LIN {X 0,Y 360.468,Z 628.216,A -85,B 0,C 180,E1 10514.88,E2 10514.88} C_VEL
LIN {X 0,Y 363.596,Z 608.418,A -85,B 0,C 180,E1 10513.753,E2 10513.753} C_VEL
LIN {X 0,Y 366.168,Z 587.631,A -85,B 0,C 180,E1 10512.86,E2 10512.86} C_VEL
LIN {X 0,Y 368.061,Z 565.565,A -85,B 0,C 180,E1 10512.202,E2 10512.202} C_VEL
LIN {X 0,Y 378.69,Z 362.963,A -85,B 0,C 180,E1 10508.029,E2 10508.029} C_VEL
LIN {X 0,Y 367.99,Z 344.813,A -85,B 0,C 180,E1 10505.531,E2 10505.531} C_VEL
LIN {X 0,Y 357.88,Z 329.138,A -85,B 0,C 180,E1 10502.966,E2 10502.966} C_VEL
LIN {X 0,Y 348.638,Z 315.938,A -85,B 0,C 180,E1 10500.418,E2 10500.418} C_VEL
LIN {X 0,Y 341.239,Z 305.859,A -85,B 0,C 180,E1 10498.178,E2 10498.178} C_VEL
LIN {X 0,Y 336.57,Z 299.556,A -85,B 0,C 180,E1 10496.589,E2 10496.589} C_VEL
LIN {X 0,Y 334.845,Z 296.268,A -85,B 0,C 180,E1 10495.437,E2 10495.437} C_VEL
LIN {X 0,Y 332.717,Z 292.115,A -85,B 0,C 180,E1 10493.916,E2 10493.916} C_VEL
LIN {X 0,Y 330.34,Z 287.641,A -85,B 0,C 180,E1 10492.18,E2 10492.18} C_VEL
LIN {X 0,Y 328.343,Z 284.042,A -85,B 0,C 180,E1 10490.663,E2 10490.663} C_VEL
LIN {X 0,Y 327.507,Z 282.562,A -85,B 0,C 180,E1 10490.018,E2 10490.018} C_VEL
LIN {X 0,Y 325.389,Z 278.836,A -85,B 0,C 180,E1 10488.301,E2 10488.301} C_VEL
LIN {X 0,Y 324.47,Z 277.349,A -85,B 0,C 180,E1 10487.56,E2 10487.56} C_VEL
LIN {X 0,Y 322.544,Z 274.367,A -85,B 0,C 180,E1 10485.984,E2 10485.984} C_VEL
LIN {X 0,Y 322.131,Z 272.803,A -85,B 0,C 180,E1 10485.207,E2 10485.207} C_VEL
LIN {X 0,Y 322.095,Z 272.581,A -85,B 0,C 180,E1 10480.765,E2 10480.765} C_VEL
LIN {X 0,Y 322.099,Z 272.578,A -85,B 0,C 180,E1 10476.361,E2 10476.361} C_VEL
LIN {X 0,Y 322.106,Z 272.587,A -85,B 0,C 180,E1 10472.058,E2 10472.058} C_VEL
LIN {X 0,Y 322.123,Z 272.61,A -85,B 0,C 180,E1 10467.747,E2 10467.747} C_VEL
LIN {X 0,Y 322.115,Z 272.598,A -85,B 0,C 180,E1 10463.215,E2 10463.215} C_VEL
LIN {X 0,Y 322.098,Z 272.579,A -85,B 0,C 180,E1 10458.784,E2 10458.784} C_VEL
LIN {X 0,Y 322.091,Z 272.575,A -85,B 0,C 180,E1 10454.378,E2 10454.378} C_VEL
LIN {X 0,Y 322.096,Z 272.592,A -85,B 0,C 180,E1 10450.009,E2 10450.009} C_VEL
LIN {X 0,Y 322.106,Z 272.613,A -85,B 0,C 180,E1 10445.699,E2 10445.699} C_VEL
LIN {X 0,Y 322.113,Z 272.591,A -85,B 0,C 180,E1 10441.244,E2 10441.244} C_VEL
LIN {X 0,Y 322.102,Z 272.579,A -85,B 0,C 180,E1 10436.796,E2 10436.796} C_VEL
LIN {X 0,Y 322.099,Z 272.578,A -85,B 0,C 180,E1 10432.507,E2 10432.507} C_VEL
LIN {X 0,Y 322.092,Z 272.584,A -85,B 0,C 180,E1 10428.176,E2 10428.176} C_VEL
LIN {X 0,Y 322.153,Z 272.865,A -85,B 0,C 180,E1 10426.904,E2 10426.904} C_VEL
LIN {X 0,Y 323.779,Z 276.577,A -85,B 0,C 180,E1 10425.147,E2 10425.147} C_VEL
LIN {X 0,Y 325.497,Z 278.631,A -85,B 0,C 180,E1 10423.95,E2 10423.95} C_VEL
LIN {X 0,Y 327.337,Z 282.289,A -85,B 0,C 180,E1 10422.397,E2 10422.397} C_VEL
LIN {X 0,Y 328.612,Z 283.991,A -85,B 0,C 180,E1 10421.551,E2 10421.551} C_VEL
LIN {X 0,Y 330.681,Z 287.818,A -85,B 0,C 180,E1 10420.02,E2 10420.02} C_VEL
LIN {X 0,Y 331.697,Z 289.424,A -85,B 0,C 180,E1 10419.347,E2 10419.347} C_VEL
LIN {X 0,Y 334.672,Z 294.855,A -85,B 0,C 180,E1 10417.33,E2 10417.33} C_VEL
LIN {X 0,Y 337.351,Z 299.62,A -85,B 0,C 180,E1 10415.67,E2 10415.67} C_VEL
LIN {X 0,Y 339.362,Z 302.724,A -85,B 0,C 180,E1 10414.76,E2 10414.76} C_VEL
LIN {X 0,Y 345.345,Z 310.607,A -85,B 0,C 180,E1 10412.87,E2 10412.87} C_VEL
LIN {X 0,Y 354.488,Z 322.89,A -85,B 0,C 180,E1 10410.236,E2 10410.236} C_VEL
LIN {X 0,Y 365.887,Z 339.496,A -85,B 0,C 180,E1 10407.242,E2 10407.242} C_VEL
LIN {X 0,Y 376.849,Z 356.898,A -85,B 0,C 180,E1 10404.615,E2 10404.615} C_VEL
LIN {X 0,Y 383.466,Z 368.195,A -85,B 0,C 180,E1 10403.129,E2 10403.129} C_VEL
LIN {X 0,Y 372.429,Z 597.085,A -85,B 0,C 180,E1 10398.572,E2 10398.572} C_VEL
LIN {X 0,Y 370.292,Z 619.591,A -85,B 0,C 180,E1 10397.939,E2 10397.939} C_VEL
LIN {X 0,Y 367.406,Z 640.687,A -85,B 0,C 180,E1 10397.111,E2 10397.111} C_VEL
LIN {X 0,Y 364.082,Z 660.164,A -85,B 0,C 180,E1 10396.094,E2 10396.094} C_VEL
LIN {X 0,Y 359.981,Z 680.411,A -85,B 0,C 180,E1 10394.754,E2 10394.754} C_VEL
LIN {X 0,Y 355.618,Z 699.418,A -85,B 0,C 180,E1 10393.203,E2 10393.203} C_VEL
LIN {X 0,Y 350.736,Z 718.51,A -85,B 0,C 180,E1 10391.293,E2 10391.293} C_VEL
LIN {X 0,Y 345.901,Z 736.013,A -85,B 0,C 180,E1 10389.165,E2 10389.165} C_VEL
LIN {X 0,Y 340.852,Z 753.347,A -85,B 0,C 180,E1 10386.649,E2 10386.649} C_VEL
LIN {X 0,Y 336.244,Z 768.991,A -85,B 0,C 180,E1 10383.938,E2 10383.938} C_VEL
LIN {X 0,Y 331.789,Z 783.986,A -85,B 0,C 180,E1 10380.81,E2 10380.81} C_VEL
LIN {X 0,Y 328.125,Z 796.845,A -85,B 0,C 180,E1 10377.59,E2 10377.59} C_VEL
LIN {X 0,Y 324.982,Z 808.929,A -85,B 0,C 180,E1 10373.959,E2 10373.959} C_VEL
LIN {X 0,Y 322.752,Z 818.965,A -85,B 0,C 180,E1 10370.3,E2 10370.3} C_VEL
LIN {X 0,Y 321.315,Z 827.026,A -85,B 0,C 180,E1 10366.633,E2 10366.633} C_VEL
LIN {X 0,Y 320.514,Z 833.651,A -85,B 0,C 180,E1 10362.794,E2 10362.794} C_VEL
LIN {X 0,Y 320.234,Z 838.371,A -85,B 0,C 180,E1 10359.161,E2 10359.161} C_VEL
LIN {X 0,Y 320.231,Z 841.275,A -85,B 0,C 180,E1 10355.732,E2 10355.732} C_VEL
LIN {X 0,Y 320.291,Z 842.922,A -85,B 0,C 180,E1 10352.324,E2 10352.324} C_VEL
LIN {X 0,Y 320.315,Z 843.073,A -85,B 0,C 180,E1 10348.925,E2 10348.925} C_VEL
LIN {X 0,Y 320.261,Z 841.954,A -85,B 0,C 180,E1 10345.522,E2 10345.522} C_VEL
LIN {X 0,Y 320.233,Z 839.199,A -85,B 0,C 180,E1 10341.921,E2 10341.921} C_VEL
LIN {X 0,Y 320.397,Z 835.01,A -85,B 0,C 180,E1 10338.295,E2 10338.295} C_VEL
LIN {X 0,Y 320.975,Z 829.102,A -85,B 0,C 180,E1 10334.644,E2 10334.644} C_VEL
LIN {X 0,Y 322.236,Z 821.155,A -85,B 0,C 180,E1 10330.796,E2 10330.796} C_VEL
LIN {X 0,Y 324.208,Z 811.793,A -85,B 0,C 180,E1 10327.132,E2 10327.132} C_VEL
LIN {X 0,Y 327.059,Z 800.358,A -85,B 0,C 180,E1 10323.489,E2 10323.489} C_VEL
LIN {X 0,Y 330.448,Z 788.162,A -85,B 0,C 180,E1 10320.248,E2 10320.248} C_VEL
LIN {X 0,Y 334.671,Z 773.926,A -85,B 0,C 180,E1 10317.06,E2 10317.06} C_VEL
LIN {X 0,Y 339.484,Z 758.214,A -85,B 0,C 180,E1 10314.118,E2 10314.118} C_VEL
LIN {X 0,Y 344.528,Z 741.355,A -85,B 0,C 180,E1 10311.499,E2 10311.499} C_VEL
LIN {X 0,Y 349.667,Z 723.67,A -85,B 0,C 180,E1 10309.201,E2 10309.201} C_VEL
LIN {X 0,Y 354.726,Z 705.255,A -85,B 0,C 180,E1 10307.209,E2 10307.209} C_VEL
LIN {X 0,Y 359.51,Z 686.034,A -85,B 0,C 180,E1 10305.503,E2 10305.503} C_VEL
LIN {X 0,Y 363.938,Z 666.085,A -85,B 0,C 180,E1 10304.074,E2 10304.074} C_VEL
LIN {X 0,Y 367.995,Z 644.8,A -85,B 0,C 180,E1 10302.866,E2 10302.866} C_VEL
LIN {X 0,Y 371.306,Z 623.779,A -85,B 0,C 180,E1 10301.96,E2 10301.96} C_VEL
LIN {X 0,Y 373.793,Z 601.62,A -85,B 0,C 180,E1 10301.28,E2 10301.28} C_VEL
LIN {X 0,Y 375.76,Z 567.676,A -85,B 0,C 180,E1 10300.547,E2 10300.547} C_VEL
LIN {X 0,Y 386.258,Z 369.62,A -85,B 0,C 180,E1 10296.548,E2 10296.548} C_VEL
LIN {X 0,Y 386.182,Z 367.946,A -85,B 0,C 180,E1 10296.479,E2 10296.479} C_VEL
LIN {X 0,Y 378.551,Z 354.327,A -85,B 0,C 180,E1 10294.374,E2 10294.374} C_VEL
LIN {X 0,Y 371.688,Z 343.11,A -85,B 0,C 180,E1 10292.275,E2 10292.275} C_VEL
LIN {X 0,Y 364.652,Z 332.437,A -85,B 0,C 180,E1 10289.847,E2 10289.847} C_VEL
LIN {X 0,Y 360.004,Z 326.055,A -85,B 0,C 180,E1 10288.04,E2 10288.04} C_VEL
LIN {X 0,Y 357.208,Z 322.172,A -85,B 0,C 180,E1 10286.832,E2 10286.832} C_VEL
LIN {X 0,Y 353.547,Z 317.389,A -85,B 0,C 180,E1 10285.102,E2 10285.102} C_VEL
LIN {X 0,Y 350.079,Z 312.934,A -85,B 0,C 180,E1 10283.213,E2 10283.213} C_VEL
LIN {X 0,Y 345.989,Z 307.675,A -85,B 0,C 180,E1 10280.468,E2 10280.468} C_VEL
LIN {X 0,Y 341.817,Z 302.664,A -85,B 0,C 180,E1 10276.485,E2 10276.485} C_VEL
LIN {X 0,Y 340.422,Z 301.286,A -85,B 0,C 180,E1 10274.242,E2 10274.242} C_VEL
LIN {X 0,Y 339.624,Z 300.553,A -85,B 0,C 180,E1 10270.004,E2 10270.004} C_VEL
LIN {X 0,Y 340.78,Z 301.638,A -85,B 0,C 180,E1 10265.895,E2 10265.895} C_VEL
LIN {X 0,Y 341.706,Z 302.868,A -85,B 0,C 180,E1 10264.533,E2 10264.533} C_VEL
LIN {X 0,Y 345.64,Z 307.471,A -85,B 0,C 180,E1 10260.664,E2 10260.664} C_VEL
LIN {X 0,Y 350.758,Z 314.248,A -85,B 0,C 180,E1 10257.224,E2 10257.224} C_VEL
LIN {X 0,Y 354.635,Z 319.419,A -85,B 0,C 180,E1 10255.149,E2 10255.149} C_VEL
LIN {X 0,Y 358.015,Z 323.91,A -85,B 0,C 180,E1 10253.587,E2 10253.587} C_VEL
LIN {X 0,Y 362.87,Z 330.765,A -85,B 0,C 180,E1 10251.577,E2 10251.577} C_VEL
LIN {X 0,Y 369.574,Z 340.739,A -85,B 0,C 180,E1 10249.14,E2 10249.14} C_VEL
LIN {X 0,Y 377.173,Z 353.186,A -85,B 0,C 180,E1 10246.706,E2 10246.706} C_VEL
LIN {X 0,Y 384.579,Z 366.332,A -85,B 0,C 180,E1 10244.585,E2 10244.585} C_VEL
LIN {X 0,Y 376.081,Z 504.545,A -85,B 0,C 180,E1 10241.656,E2 10241.656} C_VEL
LIN {X 0,Y 371.745,Z 574.559,A -85,B 0,C 180,E1 10240.129,E2 10240.129} C_VEL
LIN {X 0,Y 369.538,Z 595.372,A -85,B 0,C 180,E1 10239.421,E2 10239.421} C_VEL
LIN {X 0,Y 366.762,Z 614.562,A -85,B 0,C 180,E1 10238.523,E2 10238.523} C_VEL
LIN {X 0,Y 363.11,Z 634.83,A -85,B 0,C 180,E1 10237.29,E2 10237.29} C_VEL
LIN {X 0,Y 359.067,Z 653.718,A -85,B 0,C 180,E1 10235.839,E2 10235.839} C_VEL
LIN {X 0,Y 354.556,Z 671.965,A -85,B 0,C 180,E1 10234.106,E2 10234.106} C_VEL
LIN {X 0,Y 349.627,Z 689.677,A -85,B 0,C 180,E1 10232.032,E2 10232.032} C_VEL
LIN {X 0,Y 344.832,Z 705.493,A -85,B 0,C 180,E1 10229.779,E2 10229.779} C_VEL
LIN {X 0,Y 340.065,Z 720.299,A -85,B 0,C 180,E1 10227.237,E2 10227.237} C_VEL
LIN {X 0,Y 335.426,Z 734.252,A -85,B 0,C 180,E1 10224.329,E2 10224.329} C_VEL
LIN {X 0,Y 331.408,Z 746.244,A -85,B 0,C 180,E1 10221.293,E2 10221.293} C_VEL
LIN {X 0,Y 327.99,Z 756.708,A -85,B 0,C 180,E1 10218.06,E2 10218.06} C_VEL
LIN {X 0,Y 325.105,Z 765.978,A -85,B 0,C 180,E1 10214.481,E2 10214.481} C_VEL
LIN {X 0,Y 323.1,Z 773.069,A -85,B 0,C 180,E1 10210.971,E2 10210.971} C_VEL
LIN {X 0,Y 321.734,Z 778.689,A -85,B 0,C 180,E1 10207.294,E2 10207.294} C_VEL
LIN {X 0,Y 320.947,Z 782.735,A -85,B 0,C 180,E1 10203.466,E2 10203.466} C_VEL
LIN {X 0,Y 320.617,Z 784.964,A -85,B 0,C 180,E1 10199.898,E2 10199.898} C_VEL
LIN {X 0,Y 320.503,Z 785.677,A -85,B 0,C 180,E1 10196.453,E2 10196.453} C_VEL
LIN {X 0,Y 320.535,Z 784.98,A -85,B 0,C 180,E1 10192.951,E2 10192.951} C_VEL
LIN {X 0,Y 320.773,Z 782.771,A -85,B 0,C 180,E1 10189.295,E2 10189.295} C_VEL
LIN {X 0,Y 321.34,Z 779.074,A -85,B 0,C 180,E1 10185.708,E2 10185.708} C_VEL
LIN {X 0,Y 322.444,Z 773.454,A -85,B 0,C 180,E1 10181.993,E2 10181.993} C_VEL
LIN {X 0,Y 324.1,Z 766.47,A -85,B 0,C 180,E1 10178.518,E2 10178.518} C_VEL
LIN {X 0,Y 326.457,Z 757.782,A -85,B 0,C 180,E1 10175.098,E2 10175.098} C_VEL
LIN {X 0,Y 329.387,Z 747.821,A -85,B 0,C 180,E1 10171.915,E2 10171.915} C_VEL
LIN {X 0,Y 333.026,Z 735.918,A -85,B 0,C 180,E1 10168.798,E2 10168.798} C_VEL
LIN {X 0,Y 337.11,Z 722.518,A -85,B 0,C 180,E1 10165.92,E2 10165.92} C_VEL
LIN {X 0,Y 341.527,Z 707.629,A -85,B 0,C 180,E1 10163.277,E2 10163.277} C_VEL
LIN {X 0,Y 346.026,Z 691.721,A -85,B 0,C 180,E1 10160.941,E2 10160.941} C_VEL
LIN {X 0,Y 350.594,Z 674.213,A -85,B 0,C 180,E1 10158.817,E2 10158.817} C_VEL
LIN {X 0,Y 354.801,Z 656.509,A -85,B 0,C 180,E1 10157.056,E2 10157.056} C_VEL
LIN {X 0,Y 358.668,Z 638.055,A -85,B 0,C 180,E1 10155.554,E2 10155.554} C_VEL
LIN {X 0,Y 360.468,Z 628.216,A -85,B 0,C 180,E1 10154.88,E2 10154.88} C_VEL
LIN {X 0,Y 360.943,Z 621.249,A -85,B 0,C 180,E1 10154.34,E2 10154.34} C_VEL
LIN {X 0,Y 359.234,Z 603.834,A -85,B 0,C 180,E1 10152.764,E2 10152.764} C_VEL
LIN {X 0,Y 359.396,Z 596.605,A -85,B 0,C 180,E1 10152.324,E2 10152.324} C_VEL
LIN {X 0,Y 361.574,Z 576.065,A -85,B 0,C 180,E1 10151.595,E2 10151.595} C_VEL
LIN {X 0,Y 363.4,Z 547.671,A -85,B 0,C 180,E1 10150.929,E2 10150.929} C_VEL
LIN {X 0,Y 373.265,Z 366.495,A -85,B 0,C 180,E1 10147.185,E2 10147.185} C_VEL
LIN {X 0,Y 362.855,Z 348.784,A -85,B 0,C 180,E1 10144.659,E2 10144.659} C_VEL
LIN {X 0,Y 351.779,Z 331.567,A -85,B 0,C 180,E1 10141.718,E2 10141.718} C_VEL
LIN {X 0,Y 341.761,Z 317.456,A -85,B 0,C 180,E1 10138.779,E2 10138.779} C_VEL
LIN {X 0,Y 334.733,Z 307.973,A -85,B 0,C 180,E1 10136.521,E2 10136.521} C_VEL
LIN {X 0,Y 328.533,Z 299.676,A -85,B 0,C 180,E1 10134.247,E2 10134.247} C_VEL
LIN {X 0,Y 325.219,Z 293.589,A -85,B 0,C 180,E1 10131.836,E2 10131.836} C_VEL
LIN {X 0,Y 322.832,Z 289.018,A -85,B 0,C 180,E1 10129.897,E2 10129.897} C_VEL
LIN {X 0,Y 320.652,Z 285.352,A -85,B 0,C 180,E1 10128.144,E2 10128.144} C_VEL
LIN {X 0,Y 319.97,Z 283.961,A -85,B 0,C 180,E1 10127.513,E2 10127.513} C_VEL
LIN {X 0,Y 317.83,Z 280.648,A -85,B 0,C 180,E1 10125.706,E2 10125.706} C_VEL
LIN {X 0,Y 316.888,Z 278.672,A -85,B 0,C 180,E1 10124.715,E2 10124.715} C_VEL
LIN {X 0,Y 314.58,Z 275.328,A -85,B 0,C 180,E1 10122.607,E2 10122.607} C_VEL
LIN {X 0,Y 314.197,Z 273.735,A -85,B 0,C 180,E1 10121.687,E2 10121.687} C_VEL
LIN {X 0,Y 314.166,Z 273.575,A -85,B 0,C 180,E1 10117.288,E2 10117.288} C_VEL
LIN {X 0,Y 314.159,Z 273.59,A -85,B 0,C 180,E1 10112.753,E2 10112.753} C_VEL
LIN {X 0,Y 314.166,Z 273.598,A -85,B 0,C 180,E1 10108.305,E2 10108.305} C_VEL
LIN {X 0,Y 314.172,Z 273.574,A -85,B 0,C 180,E1 10103.838,E2 10103.838} C_VEL
LIN {X 0,Y 314.171,Z 273.561,A -85,B 0,C 180,E1 10099.52,E2 10099.52} C_VEL
LIN {X 0,Y 314.178,Z 273.567,A -85,B 0,C 180,E1 10095.125,E2 10095.125} C_VEL
LIN {X 0,Y 314.159,Z 273.594,A -85,B 0,C 180,E1 10090.636,E2 10090.636} C_VEL
LIN {X 0,Y 314.154,Z 273.592,A -85,B 0,C 180,E1 10086.211,E2 10086.211} C_VEL
LIN {X 0,Y 314.164,Z 273.573,A -85,B 0,C 180,E1 10081.64,E2 10081.64} C_VEL
LIN {X 0,Y 314.167,Z 273.564,A -85,B 0,C 180,E1 10077.262,E2 10077.262} C_VEL
LIN {X 0,Y 314.182,Z 273.565,A -85,B 0,C 180,E1 10072.869,E2 10072.869} C_VEL
LIN {X 0,Y 314.208,Z 273.926,A -85,B 0,C 180,E1 10070.382,E2 10070.382} C_VEL
LIN {X 0,Y 315.908,Z 277.658,A -85,B 0,C 180,E1 10068.312,E2 10068.312} C_VEL
LIN {X 0,Y 317.543,Z 279.349,A -85,B 0,C 180,E1 10067.08,E2 10067.08} C_VEL
LIN {X 0,Y 319.108,Z 282.876,A -85,B 0,C 180,E1 10065.482,E2 10065.482} C_VEL
LIN {X 0,Y 320.816,Z 284.892,A -85,B 0,C 180,E1 10064.266,E2 10064.266} C_VEL
LIN {X 0,Y 322.876,Z 288.899,A -85,B 0,C 180,E1 10062.518,E2 10062.518} C_VEL
LIN {X 0,Y 323.888,Z 290.291,A -85,B 0,C 180,E1 10061.832,E2 10061.832} C_VEL
LIN {X 0,Y 326.227,Z 294.454,A -85,B 0,C 180,E1 10060.109,E2 10060.109} C_VEL
LIN {X 0,Y 329.95,Z 301.234,A -85,B 0,C 180,E1 10057.552,E2 10057.552} C_VEL
LIN {X 0,Y 338.183,Z 311.866,A -85,B 0,C 180,E1 10054.707,E2 10054.707} C_VEL
LIN {X 0,Y 345.131,Z 321.016,A -85,B 0,C 180,E1 10052.524,E2 10052.524} C_VEL
LIN {X 0,Y 356.313,Z 336.923,A -85,B 0,C 180,E1 10049.334,E2 10049.334} C_VEL
LIN {X 0,Y 366.176,Z 351.963,A -85,B 0,C 180,E1 10046.782,E2 10046.782} C_VEL
LIN {X 0,Y 377.332,Z 370.289,A -85,B 0,C 180,E1 10044.13,E2 10044.13} C_VEL
LIN {X 0,Y 377.998,Z 371.985,A -85,B 0,C 180,E1 10043.962,E2 10043.962} C_VEL
LIN {X 0,Y 366.529,Z 599.992,A -85,B 0,C 180,E1 10039.376,E2 10039.376} C_VEL
LIN {X 0,Y 364.201,Z 621.903,A -85,B 0,C 180,E1 10038.721,E2 10038.721} C_VEL
LIN {X 0,Y 361.044,Z 643.25,A -85,B 0,C 180,E1 10037.838,E2 10037.838} C_VEL
LIN {X 0,Y 357.365,Z 663.639,A -85,B 0,C 180,E1 10036.726,E2 10036.726} C_VEL
LIN {X 0,Y 352.974,Z 683.917,A -85,B 0,C 180,E1 10035.313,E2 10035.313} C_VEL
LIN {X 0,Y 348.283,Z 703.006,A -85,B 0,C 180,E1 10033.659,E2 10033.659} C_VEL
LIN {X 0,Y 343.101,Z 722.188,A -85,B 0,C 180,E1 10031.636,E2 10031.636} C_VEL
LIN {X 0,Y 337.996,Z 739.862,A -85,B 0,C 180,E1 10029.383,E2 10029.383} C_VEL
LIN {X 0,Y 332.867,Z 756.479,A -85,B 0,C 180,E1 10026.814,E2 10026.814} C_VEL
LIN {X 0,Y 327.963,Z 772.177,A -85,B 0,C 180,E1 10023.909,E2 10023.909} C_VEL
LIN {X 0,Y 323.638,Z 786.221,A -85,B 0,C 180,E1 10020.81,E2 10020.81} C_VEL
LIN {X 0,Y 319.801,Z 799.27,A -85,B 0,C 180,E1 10017.359,E2 10017.359} C_VEL
LIN {X 0,Y 316.775,Z 810.476,A -85,B 0,C 180,E1 10013.743,E2 10013.743} C_VEL
LIN {X 0,Y 314.525,Z 820.295,A -85,B 0,C 180,E1 10009.884,E2 10009.884} C_VEL
LIN {X 0,Y 313.145,Z 828.175,A -85,B 0,C 180,E1 10006.036,E2 10006.036} C_VEL
LIN {X 0,Y 312.469,Z 833.97,A -85,B 0,C 180,E1 10002.378,E2 10002.378} C_VEL
LIN {X 0,Y 312.239,Z 838.49,A -85,B 0,C 180,E1 9998.469,E2 9998.469} C_VEL
LIN {X 0,Y 312.272,Z 841.025,A -85,B 0,C 180,E1 9995.142,E2 9995.142} C_VEL
LIN {X 0,Y 312.337,Z 842.339,A -85,B 0,C 180,E1 9991.466,E2 9991.466} C_VEL
LIN {X 0,Y 312.34,Z 842.269,A -85,B 0,C 180,E1 9988.347,E2 9988.347} C_VEL
LIN {X 0,Y 312.274,Z 840.796,A -85,B 0,C 180,E1 9984.67,E2 9984.67} C_VEL
LIN {X 0,Y 312.248,Z 838.123,A -85,B 0,C 180,E1 9981.342,E2 9981.342} C_VEL
LIN {X 0,Y 312.496,Z 833.458,A -85,B 0,C 180,E1 9977.432,E2 9977.432} C_VEL
LIN {X 0,Y 313.217,Z 827.376,A -85,B 0,C 180,E1 9973.683,E2 9973.683} C_VEL
LIN {X 0,Y 314.597,Z 819.539,A -85,B 0,C 180,E1 9969.923,E2 9969.923} C_VEL
LIN {X 0,Y 316.807,Z 809.959,A -85,B 0,C 180,E1 9966.171,E2 9966.171} C_VEL
LIN {X 0,Y 319.956,Z 798.388,A -85,B 0,C 180,E1 9962.45,E2 9962.45} C_VEL
LIN {X 0,Y 323.894,Z 785.209,A -85,B 0,C 180,E1 9958.965,E2 9958.965} C_VEL
LIN {X 0,Y 328.528,Z 770.539,A -85,B 0,C 180,E1 9955.732,E2 9955.732} C_VEL
LIN {X 0,Y 333.415,Z 755.305,A -85,B 0,C 180,E1 9952.911,E2 9952.911} C_VEL
LIN {X 0,Y 338.815,Z 738.345,A -85,B 0,C 180,E1 9950.288,E2 9950.288} C_VEL
LIN {X 0,Y 344.045,Z 720.877,A -85,B 0,C 180,E1 9948.053,E2 9948.053} C_VEL
LIN {X 0,Y 349.591,Z 701.225,A -85,B 0,C 180,E1 9945.971,E2 9945.971} C_VEL
LIN {X 0,Y 354.435,Z 682.492,A -85,B 0,C 180,E1 9944.345,E2 9944.345} C_VEL
LIN {X 0,Y 358.824,Z 663.098,A -85,B 0,C 180,E1 9942.99,E2 9942.99} C_VEL
LIN {X 0,Y 362.799,Z 642.542,A -85,B 0,C 180,E1 9941.852,E2 9941.852} C_VEL
LIN {X 0,Y 366.132,Z 621.734,A -85,B 0,C 180,E1 9940.973,E2 9940.973} C_VEL
LIN {X 0,Y 368.657,Z 599.714,A -85,B 0,C 180,E1 9940.302,E2 9940.302} C_VEL
LIN {X 0,Y 371.066,Z 557.618,A -85,B 0,C 180,E1 9939.408,E2 9939.408} C_VEL
LIN {X 0,Y 381.414,Z 371.832,A -85,B 0,C 180,E1 9935.613,E2 9935.613} C_VEL
LIN {X 0,Y 373.499,Z 357.554,A -85,B 0,C 180,E1 9933.285,E2 9933.285} C_VEL
LIN {X 0,Y 366.412,Z 346.056,A -85,B 0,C 180,E1 9930.957,E2 9930.957} C_VEL
LIN {X 0,Y 359.26,Z 335.206,A -85,B 0,C 180,E1 9928.238,E2 9928.238} C_VEL
LIN {X 0,Y 354.734,Z 329.033,A -85,B 0,C 180,E1 9926.266,E2 9926.266} C_VEL
LIN {X 0,Y 351.472,Z 324.589,A -85,B 0,C 180,E1 9924.631,E2 9924.631} C_VEL
LIN {X 0,Y 348.234,Z 320.367,A -85,B 0,C 180,E1 9922.807,E2 9922.807} C_VEL
LIN {X 0,Y 344.522,Z 315.397,A -85,B 0,C 180,E1 9920.205,E2 9920.205} C_VEL
LIN {X 0,Y 340.156,Z 309.887,A -85,B 0,C 180,E1 9915.691,E2 9915.691} C_VEL
LIN {X 0,Y 338.403,Z 308.486,A -85,B 0,C 180,E1 9911.246,E2 9911.246} C_VEL
LIN {X 0,Y 338.951,Z 308.966,A -85,B 0,C 180,E1 9907.459,E2 9907.459} C_VEL
LIN {X 0,Y 340.26,Z 310.296,A -85,B 0,C 180,E1 9905.013,E2 9905.013} C_VEL
LIN {X 0,Y 344.075,Z 315.129,A -85,B 0,C 180,E1 9901,E2 9901} C_VEL
LIN {X 0,Y 348.896,Z 321.642,A -85,B 0,C 180,E1 9897.62,E2 9897.62} C_VEL
LIN {X 0,Y 352.723,Z 326.935,A -85,B 0,C 180,E1 9895.49,E2 9895.49} C_VEL
LIN {X 0,Y 355.865,Z 331.23,A -85,B 0,C 180,E1 9893.99,E2 9893.99} C_VEL
LIN {X 0,Y 360.991,Z 338.617,A -85,B 0,C 180,E1 9891.801,E2 9891.801} C_VEL
LIN {X 0,Y 368.01,Z 349.59,A -85,B 0,C 180,E1 9889.196,E2 9889.196} C_VEL
LIN {X 0,Y 375.731,Z 362.654,A -85,B 0,C 180,E1 9886.694,E2 9886.694} C_VEL
LIN {X 0,Y 379.861,Z 370.595,A -85,B 0,C 180,E1 9885.455,E2 9885.455} C_VEL
LIN {X 0,Y 366.599,Z 574.331,A -85,B 0,C 180,E1 9881.089,E2 9881.089} C_VEL
LIN {X 0,Y 364.339,Z 594.972,A -85,B 0,C 180,E1 9880.389,E2 9880.389} C_VEL
LIN {X 0,Y 361.383,Z 614.906,A -85,B 0,C 180,E1 9879.46,E2 9879.46} C_VEL
LIN {X 0,Y 357.527,Z 635.514,A -85,B 0,C 180,E1 9878.2,E2 9878.2} C_VEL
LIN {X 0,Y 353.365,Z 654.14,A -85,B 0,C 180,E1 9876.757,E2 9876.757} C_VEL
LIN {X 0,Y 348.63,Z 672.487,A -85,B 0,C 180,E1 9874.998,E2 9874.998} C_VEL
LIN {X 0,Y 343.569,Z 689.916,A -85,B 0,C 180,E1 9872.942,E2 9872.942} C_VEL
LIN {X 0,Y 338.488,Z 705.939,A -85,B 0,C 180,E1 9870.639,E2 9870.639} C_VEL
LIN {X 0,Y 333.462,Z 720.789,A -85,B 0,C 180,E1 9868.057,E2 9868.057} C_VEL
LIN {X 0,Y 328.582,Z 734.758,A -85,B 0,C 180,E1 9865.107,E2 9865.107} C_VEL
LIN {X 0,Y 324.415,Z 746.511,A -85,B 0,C 180,E1 9862.094,E2 9862.094} C_VEL
LIN {X 0,Y 320.666,Z 757.265,A -85,B 0,C 180,E1 9858.719,E2 9858.719} C_VEL
LIN {X 0,Y 317.599,Z 766.459,A -85,B 0,C 180,E1 9855.102,E2 9855.102} C_VEL
LIN {X 0,Y 315.415,Z 773.626,A -85,B 0,C 180,E1 9851.495,E2 9851.495} C_VEL
LIN {X 0,Y 313.91,Z 779.317,A -85,B 0,C 180,E1 9847.704,E2 9847.704} C_VEL
LIN {X 0,Y 313.035,Z 783.41,A -85,B 0,C 180,E1 9843.766,E2 9843.766} C_VEL
LIN {X 0,Y 312.667,Z 785.659,A -85,B 0,C 180,E1 9840.138,E2 9840.138} C_VEL
LIN {X 0,Y 312.537,Z 786.389,A -85,B 0,C 180,E1 9836.61,E2 9836.61} C_VEL
LIN {X 0,Y 312.571,Z 785.694,A -85,B 0,C 180,E1 9832.895,E2 9832.895} C_VEL
LIN {X 0,Y 312.82,Z 783.544,A -85,B 0,C 180,E1 9829.223,E2 9829.223} C_VEL
LIN {X 0,Y 313.421,Z 779.865,A -85,B 0,C 180,E1 9825.545,E2 9825.545} C_VEL
LIN {X 0,Y 314.592,Z 774.273,A -85,B 0,C 180,E1 9821.738,E2 9821.738} C_VEL
LIN {X 0,Y 316.345,Z 767.329,A -85,B 0,C 180,E1 9818.179,E2 9818.179} C_VEL
LIN {X 0,Y 318.984,Z 758.173,A -85,B 0,C 180,E1 9814.496,E2 9814.496} C_VEL
LIN {X 0,Y 322.294,Z 747.519,A -85,B 0,C 180,E1 9811.068,E2 9811.068} C_VEL
LIN {X 0,Y 325.956,Z 736.16,A -85,B 0,C 180,E1 9808.068,E2 9808.068} C_VEL
LIN {X 0,Y 330.268,Z 722.698,A -85,B 0,C 180,E1 9805.139,E2 9805.139} C_VEL
LIN {X 0,Y 334.913,Z 707.697,A -85,B 0,C 180,E1 9802.454,E2 9802.454} C_VEL
LIN {X 0,Y 339.45,Z 692.267,A -85,B 0,C 180,E1 9800.165,E2 9800.165} C_VEL
LIN {X 0,Y 344.206,Z 674.76,A -85,B 0,C 180,E1 9798.015,E2 9798.015} C_VEL
LIN {X 0,Y 348.588,Z 657.018,A -85,B 0,C 180,E1 9796.229,E2 9796.229} C_VEL
LIN {X 0,Y 352.603,Z 638.551,A -85,B 0,C 180,E1 9794.711,E2 9794.711} C_VEL
LIN {X 0,Y 356.321,Z 617.92,A -85,B 0,C 180,E1 9793.37,E2 9793.37} C_VEL
LIN {X 0,Y 359.296,Z 597.325,A -85,B 0,C 180,E1 9792.355,E2 9792.355} C_VEL
LIN {X 0,Y 359.396,Z 596.605,A -85,B 0,C 180,E1 9792.324,E2 9792.324} C_VEL
LIN {X 0,Y 359.58,Z 589.279,A -85,B 0,C 180,E1 9791.911,E2 9791.911} C_VEL
LIN {X 0,Y 357.119,Z 570.935,A -85,B 0,C 180,E1 9790.654,E2 9790.654} C_VEL
LIN {X 0,Y 356.908,Z 563.421,A -85,B 0,C 180,E1 9790.355,E2 9790.355} C_VEL
LIN {X 0,Y 367.921,Z 370.065,A -85,B 0,C 180,E1 9786.318,E2 9786.318} C_VEL
LIN {X 0,Y 358.108,Z 353.301,A -85,B 0,C 180,E1 9783.845,E2 9783.845} C_VEL
LIN {X 0,Y 347.995,Z 337.495,A -85,B 0,C 180,E1 9781.07,E2 9781.07} C_VEL
LIN {X 0,Y 338.371,Z 323.742,A -85,B 0,C 180,E1 9778.157,E2 9778.157} C_VEL
LIN {X 0,Y 331.127,Z 313.838,A -85,B 0,C 180,E1 9775.748,E2 9775.748} C_VEL
LIN {X 0,Y 324.221,Z 304.961,A -85,B 0,C 180,E1 9773.226,E2 9773.226} C_VEL
LIN {X 0,Y 320.37,Z 299.828,A -85,B 0,C 180,E1 9771.609,E2 9771.609} C_VEL
LIN {X 0,Y 317.855,Z 295.123,A -85,B 0,C 180,E1 9769.571,E2 9769.571} C_VEL
LIN {X 0,Y 315.671,Z 291.109,A -85,B 0,C 180,E1 9767.693,E2 9767.693} C_VEL
LIN {X 0,Y 312.926,Z 286.361,A -85,B 0,C 180,E1 9765.178,E2 9765.178} C_VEL
LIN {X 0,Y 311.992,Z 284.881,A -85,B 0,C 180,E1 9764.315,E2 9764.315} C_VEL
LIN {X 0,Y 309.872,Z 281.344,A -85,B 0,C 180,E1 9762.153,E2 9762.153} C_VEL
LIN {X 0,Y 309.154,Z 279.823,A -85,B 0,C 180,E1 9761.28,E2 9761.28} C_VEL
LIN {X 0,Y 306.603,Z 276.218,A -85,B 0,C 180,E1 9758.499,E2 9758.499} C_VEL
LIN {X 0,Y 306.249,Z 274.709,A -85,B 0,C 180,E1 9757.389,E2 9757.389} C_VEL
LIN {X 0,Y 306.221,Z 274.579,A -85,B 0,C 180,E1 9752.819,E2 9752.819} C_VEL
LIN {X 0,Y 306.23,Z 274.586,A -85,B 0,C 180,E1 9748.255,E2 9748.255} C_VEL
LIN {X 0,Y 306.236,Z 274.564,A -85,B 0,C 180,E1 9743.676,E2 9743.676} C_VEL
LIN {X 0,Y 306.23,Z 274.55,A -85,B 0,C 180,E1 9739.253,E2 9739.253} C_VEL
LIN {X 0,Y 306.22,Z 274.553,A -85,B 0,C 180,E1 9734.753,E2 9734.753} C_VEL
LIN {X 0,Y 306.217,Z 274.57,A -85,B 0,C 180,E1 9730.154,E2 9730.154} C_VEL
LIN {X 0,Y 306.23,Z 274.592,A -85,B 0,C 180,E1 9725.62,E2 9725.62} C_VEL
LIN {X 0,Y 306.237,Z 274.568,A -85,B 0,C 180,E1 9721.121,E2 9721.121} C_VEL
LIN {X 0,Y 306.22,Z 274.557,A -85,B 0,C 180,E1 9716.629,E2 9716.629} C_VEL
LIN {X 0,Y 306.275,Z 274.934,A -85,B 0,C 180,E1 9714.566,E2 9714.566} C_VEL
LIN {X 0,Y 308.125,Z 278.831,A -85,B 0,C 180,E1 9711.978,E2 9711.978} C_VEL
LIN {X 0,Y 309.742,Z 280.576,A -85,B 0,C 180,E1 9710.523,E2 9710.523} C_VEL
LIN {X 0,Y 311.72,Z 284.506,A -85,B 0,C 180,E1 9708.34,E2 9708.34} C_VEL
LIN {X 0,Y 313.075,Z 286.025,A -85,B 0,C 180,E1 9707.268,E2 9707.268} C_VEL
LIN {X 0,Y 314.893,Z 289.76,A -85,B 0,C 180,E1 9705.471,E2 9705.471} C_VEL
LIN {X 0,Y 316.303,Z 291.631,A -85,B 0,C 180,E1 9704.412,E2 9704.412} C_VEL
LIN {X 0,Y 318.675,Z 295.813,A -85,B 0,C 180,E1 9702.469,E2 9702.469} C_VEL
LIN {X 0,Y 322.238,Z 301.811,A -85,B 0,C 180,E1 9699.995,E2 9699.995} C_VEL
LIN {X 0,Y 326.055,Z 306.59,A -85,B 0,C 180,E1 9698.502,E2 9698.502} C_VEL
LIN {X 0,Y 335.614,Z 319.134,A -85,B 0,C 180,E1 9695.113,E2 9695.113} C_VEL
LIN {X 0,Y 342.247,Z 328.046,A -85,B 0,C 180,E1 9692.98,E2 9692.98} C_VEL
LIN {X 0,Y 352.812,Z 343.235,A -85,B 0,C 180,E1 9689.892,E2 9689.892} C_VEL
LIN {X 0,Y 362.621,Z 358.408,A -85,B 0,C 180,E1 9687.286,E2 9687.286} C_VEL
LIN {X 0,Y 372.652,Z 375.063,A -85,B 0,C 180,E1 9684.833,E2 9684.833} C_VEL
LIN {X 0,Y 360.85,Z 599.921,A -85,B 0,C 180,E1 9680.268,E2 9680.268} C_VEL
LIN {X 0,Y 358.42,Z 622.01,A -85,B 0,C 180,E1 9679.599,E2 9679.599} C_VEL
LIN {X 0,Y 355.206,Z 642.991,A -85,B 0,C 180,E1 9678.723,E2 9678.723} C_VEL
LIN {X 0,Y 351.627,Z 662.354,A -85,B 0,C 180,E1 9677.67,E2 9677.67} C_VEL
LIN {X 0,Y 347.148,Z 682.462,A -85,B 0,C 180,E1 9676.27,E2 9676.27} C_VEL
LIN {X 0,Y 342.087,Z 702.377,A -85,B 0,C 180,E1 9674.542,E2 9674.542} C_VEL
LIN {X 0,Y 336.904,Z 720.891,A -85,B 0,C 180,E1 9672.58,E2 9672.58} C_VEL
LIN {X 0,Y 331.477,Z 738.948,A -85,B 0,C 180,E1 9670.257,E2 9670.257} C_VEL
LIN {X 0,Y 326.318,Z 754.965,A -85,B 0,C 180,E1 9667.764,E2 9667.764} C_VEL
LIN {X 0,Y 321.041,Z 771.173,A -85,B 0,C 180,E1 9664.743,E2 9664.743} C_VEL
LIN {X 0,Y 316.509,Z 785.132,A -85,B 0,C 180,E1 9661.625,E2 9661.625} C_VEL
LIN {X 0,Y 312.582,Z 797.689,A -85,B 0,C 180,E1 9658.253,E2 9658.253} C_VEL
LIN {X 0,Y 309.359,Z 808.845,A -85,B 0,C 180,E1 9654.639,E2 9654.639} C_VEL
LIN {X 0,Y 306.929,Z 818.663,A -85,B 0,C 180,E1 9650.78,E2 9650.78} C_VEL
LIN {X 0,Y 305.384,Z 826.559,A -85,B 0,C 180,E1 9646.939,E2 9646.939} C_VEL
LIN {X 0,Y 304.56,Z 832.667,A -85,B 0,C 180,E1 9643.09,E2 9643.09} C_VEL
LIN {X 0,Y 304.27,Z 837.24,A -85,B 0,C 180,E1 9639.264,E2 9639.264} C_VEL
LIN {X 0,Y 304.282,Z 840.058,A -85,B 0,C 180,E1 9635.655,E2 9635.655} C_VEL
LIN {X 0,Y 304.363,Z 841.579,A -85,B 0,C 180,E1 9631.881,E2 9631.881} C_VEL
LIN {X 0,Y 304.375,Z 841.615,A -85,B 0,C 180,E1 9628.68,E2 9628.68} C_VEL
LIN {X 0,Y 304.306,Z 840.437,A -85,B 0,C 180,E1 9625.097,E2 9625.097} C_VEL
LIN {X 0,Y 304.265,Z 837.757,A -85,B 0,C 180,E1 9621.494,E2 9621.494} C_VEL
LIN {X 0,Y 304.473,Z 833.553,A -85,B 0,C 180,E1 9617.673,E2 9617.673} C_VEL
LIN {X 0,Y 305.199,Z 827.447,A -85,B 0,C 180,E1 9613.72,E2 9613.72} C_VEL
LIN {X 0,Y 306.73,Z 819.239,A -85,B 0,C 180,E1 9609.585,E2 9609.585} C_VEL
LIN {X 0,Y 309.058,Z 809.76,A -85,B 0,C 180,E1 9605.739,E2 9605.739} C_VEL
LIN {X 0,Y 312.373,Z 798.261,A -85,B 0,C 180,E1 9601.93,E2 9601.93} C_VEL
LIN {X 0,Y 316.264,Z 785.942,A -85,B 0,C 180,E1 9598.556,E2 9598.556} C_VEL
LIN {X 0,Y 321.067,Z 771.574,A -85,B 0,C 180,E1 9595.255,E2 9595.255} C_VEL
LIN {X 0,Y 326.268,Z 756.258,A -85,B 0,C 180,E1 9592.309,E2 9592.309} C_VEL
LIN {X 0,Y 331.883,Z 739.352,A -85,B 0,C 180,E1 9589.628,E2 9589.628} C_VEL
LIN {X 0,Y 337.517,Z 721.581,A -85,B 0,C 180,E1 9587.28,E2 9587.28} C_VEL
LIN {X 0,Y 343.04,Z 703.048,A -85,B 0,C 180,E1 9585.257,E2 9585.257} C_VEL
LIN {X 0,Y 348.525,Z 682.857,A -85,B 0,C 180,E1 9583.462,E2 9583.462} C_VEL
LIN {X 0,Y 353.284,Z 662.693,A -85,B 0,C 180,E1 9582.037,E2 9582.037} C_VEL
LIN {X 0,Y 357.434,Z 642.07,A -85,B 0,C 180,E1 9580.888,E2 9580.888} C_VEL
LIN {X 0,Y 360.866,Z 621.401,A -85,B 0,C 180,E1 9580.013,E2 9580.013} C_VEL
LIN {X 0,Y 363.499,Z 599.187,A -85,B 0,C 180,E1 9579.334,E2 9579.334} C_VEL
LIN {X 0,Y 366.082,Z 556.29,A -85,B 0,C 180,E1 9578.414,E2 9578.414} C_VEL
LIN {X 0,Y 376.685,Z 375.684,A -85,B 0,C 180,E1 9574.695,E2 9574.695} C_VEL
LIN {X 0,Y 369.886,Z 363.231,A -85,B 0,C 180,E1 9572.59,E2 9572.59} C_VEL
LIN {X 0,Y 363.241,Z 352.17,A -85,B 0,C 180,E1 9570.293,E2 9570.293} C_VEL
LIN {X 0,Y 356.8,Z 342.144,A -85,B 0,C 180,E1 9567.723,E2 9567.723} C_VEL
LIN {X 0,Y 352.57,Z 336.202,A -85,B 0,C 180,E1 9565.806,E2 9565.806} C_VEL
LIN {X 0,Y 349.277,Z 331.598,A -85,B 0,C 180,E1 9564.076,E2 9564.076} C_VEL
LIN {X 0,Y 346.564,Z 327.934,A -85,B 0,C 180,E1 9562.475,E2 9562.475} C_VEL
LIN {X 0,Y 343.063,Z 323.117,A -85,B 0,C 180,E1 9559.939,E2 9559.939} C_VEL
LIN {X 0,Y 338.896,Z 317.693,A -85,B 0,C 180,E1 9555.4,E2 9555.4} C_VEL
LIN {X 0,Y 337.319,Z 316.405,A -85,B 0,C 180,E1 9551.11,E2 9551.11} C_VEL
LIN {X 0,Y 337.929,Z 316.955,A -85,B 0,C 180,E1 9547.311,E2 9547.311} C_VEL
LIN {X 0,Y 338.998,Z 318.08,A -85,B 0,C 180,E1 9545.247,E2 9545.247} C_VEL
LIN {X 0,Y 343.138,Z 323.542,A -85,B 0,C 180,E1 9540.836,E2 9540.836} C_VEL
LIN {X 0,Y 347.448,Z 329.616,A -85,B 0,C 180,E1 9537.775,E2 9537.775} C_VEL
LIN {X 0,Y 350.896,Z 334.526,A -85,B 0,C 180,E1 9535.806,E2 9535.806} C_VEL
LIN {X 0,Y 353.717,Z 338.516,A -85,B 0,C 180,E1 9534.405,E2 9534.405} C_VEL
LIN {X 0,Y 358.616,Z 345.803,A -85,B 0,C 180,E1 9532.23,E2 9532.23} C_VEL
LIN {X 0,Y 365.781,Z 357.297,A -85,B 0,C 180,E1 9529.488,E2 9529.488} C_VEL
LIN {X 0,Y 372.952,Z 370.003,A -85,B 0,C 180,E1 9527.086,E2 9527.086} C_VEL
LIN {X 0,Y 375.144,Z 374.406,A -85,B 0,C 180,E1 9526.388,E2 9526.388} C_VEL
LIN {X 0,Y 361.507,Z 575.086,A -85,B 0,C 180,E1 9522.053,E2 9522.053} C_VEL
LIN {X 0,Y 359.136,Z 595.875,A -85,B 0,C 180,E1 9521.341,E2 9521.341} C_VEL
LIN {X 0,Y 356.102,Z 615.44,A -85,B 0,C 180,E1 9520.42,E2 9520.42} C_VEL
LIN {X 0,Y 352.31,Z 635.01,A -85,B 0,C 180,E1 9519.224,E2 9519.224} C_VEL
LIN {X 0,Y 347.88,Z 654.174,A -85,B 0,C 180,E1 9517.743,E2 9517.743} C_VEL
LIN {X 0,Y 343.072,Z 672.124,A -85,B 0,C 180,E1 9516.021,E2 9516.021} C_VEL
LIN {X 0,Y 337.98,Z 688.98,A -85,B 0,C 180,E1 9514.036,E2 9514.036} C_VEL
LIN {X 0,Y 332.648,Z 705.158,A -85,B 0,C 180,E1 9511.728,E2 9511.728} C_VEL
LIN {X 0,Y 327.363,Z 720.209,A -85,B 0,C 180,E1 9509.124,E2 9509.124} C_VEL
LIN {X 0,Y 322.384,Z 733.765,A -85,B 0,C 180,E1 9506.281,E2 9506.281} C_VEL
LIN {X 0,Y 317.649,Z 746.405,A -85,B 0,C 180,E1 9503.046,E2 9503.046} C_VEL
LIN {X 0,Y 313.508,Z 757.499,A -85,B 0,C 180,E1 9499.524,E2 9499.524} C_VEL
LIN {X 0,Y 310.229,Z 766.639,A -85,B 0,C 180,E1 9495.883,E2 9495.883} C_VEL
LIN {X 0,Y 307.851,Z 773.869,A -85,B 0,C 180,E1 9492.228,E2 9492.228} C_VEL
LIN {X 0,Y 306.17,Z 779.686,A -85,B 0,C 180,E1 9488.353,E2 9488.353} C_VEL
LIN {X 0,Y 305.209,Z 783.748,A -85,B 0,C 180,E1 9484.525,E2 9484.525} C_VEL
LIN {X 0,Y 304.743,Z 786.193,A -85,B 0,C 180,E1 9480.731,E2 9480.731} C_VEL
LIN {X 0,Y 304.572,Z 787.072,A -85,B 0,C 180,E1 9477.151,E2 9477.151} C_VEL
LIN {X 0,Y 304.588,Z 786.625,A -85,B 0,C 180,E1 9473.405,E2 9473.405} C_VEL
LIN {X 0,Y 304.808,Z 784.752,A -85,B 0,C 180,E1 9469.712,E2 9469.712} C_VEL
LIN {X 0,Y 305.367,Z 781.292,A -85,B 0,C 180,E1 9465.966,E2 9465.966} C_VEL
LIN {X 0,Y 306.511,Z 776.015,A -85,B 0,C 180,E1 9462.052,E2 9462.052} C_VEL
LIN {X 0,Y 308.372,Z 768.997,A -85,B 0,C 180,E1 9458.204,E2 9458.204} C_VEL
LIN {X 0,Y 310.938,Z 760.521,A -85,B 0,C 180,E1 9454.585,E2 9454.585} C_VEL
LIN {X 0,Y 314.266,Z 750.316,A -85,B 0,C 180,E1 9451.096,E2 9451.096} C_VEL
LIN {X 0,Y 318.208,Z 738.542,A -85,B 0,C 180,E1 9447.841,E2 9447.841} C_VEL
LIN {X 0,Y 322.627,Z 725.353,A -85,B 0,C 180,E1 9444.846,E2 9444.846} C_VEL
LIN {X 0,Y 327.395,Z 710.738,A -85,B 0,C 180,E1 9442.103,E2 9442.103} C_VEL
LIN {X 0,Y 332.415,Z 694.584,A -85,B 0,C 180,E1 9439.605,E2 9439.605} C_VEL
LIN {X 0,Y 337.141,Z 678.119,A -85,B 0,C 180,E1 9437.499,E2 9437.499} C_VEL
LIN {X 0,Y 341.848,Z 660.074,A -85,B 0,C 180,E1 9435.606,E2 9435.606} C_VEL
LIN {X 0,Y 346.179,Z 640.954,A -85,B 0,C 180,E1 9433.991,E2 9433.991} C_VEL
LIN {X 0,Y 349.804,Z 622.002,A -85,B 0,C 180,E1 9432.708,E2 9432.708} C_VEL
LIN {X 0,Y 353.11,Z 600.787,A -85,B 0,C 180,E1 9431.598,E2 9431.598} C_VEL
LIN {X 0,Y 355.649,Z 579.107,A -85,B 0,C 180,E1 9430.777,E2 9430.777} C_VEL
LIN {X 0,Y 356.908,Z 563.421,A -85,B 0,C 180,E1 9430.355,E2 9430.355} C_VEL
LIN {X 0,Y 356.709,Z 555.868,A -85,B 0,C 180,E1 9430.067,E2 9430.067} C_VEL
LIN {X 0,Y 353.517,Z 536.106,A -85,B 0,C 180,E1 9428.916,E2 9428.916} C_VEL
LIN {X 0,Y 353.374,Z 529.595,A -85,B 0,C 180,E1 9428.691,E2 9428.691} C_VEL
LIN {X 0,Y 362.502,Z 373.41,A -85,B 0,C 180,E1 9425.397,E2 9425.397} C_VEL
LIN {X 0,Y 353.517,Z 358.055,A -85,B 0,C 180,E1 9423.041,E2 9423.041} C_VEL
LIN {X 0,Y 344.365,Z 343.568,A -85,B 0,C 180,E1 9420.441,E2 9420.441} C_VEL
LIN {X 0,Y 335.178,Z 330.26,A -85,B 0,C 180,E1 9417.583,E2 9417.583} C_VEL
LIN {X 0,Y 327.456,Z 319.544,A -85,B 0,C 180,E1 9414.913,E2 9414.913} C_VEL
LIN {X 0,Y 321.469,Z 311.823,A -85,B 0,C 180,E1 9412.666,E2 9412.666} C_VEL
LIN {X 0,Y 317.298,Z 306.487,A -85,B 0,C 180,E1 9410.961,E2 9410.961} C_VEL
LIN {X 0,Y 312.793,Z 300.905,A -85,B 0,C 180,E1 9408.968,E2 9408.968} C_VEL
LIN {X 0,Y 310.249,Z 296.431,A -85,B 0,C 180,E1 9406.907,E2 9406.907} C_VEL
LIN {X 0,Y 308.124,Z 292.35,A -85,B 0,C 180,E1 9404.759,E2 9404.759} C_VEL
LIN {X 0,Y 305.286,Z 287.804,A -85,B 0,C 180,E1 9401.92,E2 9401.92} C_VEL
LIN {X 0,Y 304.58,Z 286.332,A -85,B 0,C 180,E1 9401.034,E2 9401.034} C_VEL
LIN {X 0,Y 302.115,Z 282.688,A -85,B 0,C 180,E1 9398.232,E2 9398.232} C_VEL
LIN {X 0,Y 301.456,Z 281.031,A -85,B 0,C 180,E1 9397.129,E2 9397.129} C_VEL
LIN {X 0,Y 298.627,Z 277.081,A -85,B 0,C 180,E1 9393.175,E2 9393.175} C_VEL
LIN {X 0,Y 298.31,Z 275.645,A -85,B 0,C 180,E1 9391.647,E2 9391.647} C_VEL
LIN {X 0,Y 298.292,Z 275.56,A -85,B 0,C 180,E1 9387.118,E2 9387.118} C_VEL
LIN {X 0,Y 298.283,Z 275.581,A -85,B 0,C 180,E1 9382.464,E2 9382.464} C_VEL
LIN {X 0,Y 298.29,Z 275.554,A -85,B 0,C 180,E1 9377.841,E2 9377.841} C_VEL
LIN {X 0,Y 298.296,Z 275.538,A -85,B 0,C 180,E1 9373.371,E2 9373.371} C_VEL
LIN {X 0,Y 298.286,Z 275.54,A -85,B 0,C 180,E1 9368.868,E2 9368.868} C_VEL
LIN {X 0,Y 298.277,Z 275.556,A -85,B 0,C 180,E1 9364.42,E2 9364.42} C_VEL
LIN {X 0,Y 298.316,Z 275.841,A -85,B 0,C 180,E1 9360.382,E2 9360.382} C_VEL
LIN {X 0,Y 300.784,Z 280.443,A -85,B 0,C 180,E1 9355.996,E2 9355.996} C_VEL
LIN {X 0,Y 301.978,Z 281.746,A -85,B 0,C 180,E1 9354.679,E2 9354.679} C_VEL
LIN {X 0,Y 304.114,Z 285.841,A -85,B 0,C 180,E1 9351.871,E2 9351.871} C_VEL
LIN {X 0,Y 305.33,Z 287.179,A -85,B 0,C 180,E1 9350.765,E2 9350.765} C_VEL
LIN {X 0,Y 307.288,Z 291.076,A -85,B 0,C 180,E1 9348.55,E2 9348.55} C_VEL
LIN {X 0,Y 308.579,Z 292.684,A -85,B 0,C 180,E1 9347.46,E2 9347.46} C_VEL
LIN {X 0,Y 310.675,Z 296.629,A -85,B 0,C 180,E1 9345.46,E2 9345.46} C_VEL
LIN {X 0,Y 311.798,Z 298.333,A -85,B 0,C 180,E1 9344.563,E2 9344.563} C_VEL
LIN {X 0,Y 313.971,Z 301.959,A -85,B 0,C 180,E1 9342.962,E2 9342.962} C_VEL
LIN {X 0,Y 320.104,Z 309.516,A -85,B 0,C 180,E1 9340.331,E2 9340.331} C_VEL
LIN {X 0,Y 325.793,Z 316.846,A -85,B 0,C 180,E1 9338.105,E2 9338.105} C_VEL
LIN {X 0,Y 335.115,Z 328.999,A -85,B 0,C 180,E1 9334.838,E2 9334.838} C_VEL
LIN {X 0,Y 345.62,Z 344.063,A -85,B 0,C 180,E1 9331.535,E2 9331.535} C_VEL
LIN {X 0,Y 355.007,Z 358.309,A -85,B 0,C 180,E1 9328.88,E2 9328.88} C_VEL
LIN {X 0,Y 365.066,Z 374.876,A -85,B 0,C 180,E1 9326.268,E2 9326.268} C_VEL
LIN {X 0,Y 367.303,Z 378.962,A -85,B 0,C 180,E1 9325.71,E2 9325.71} C_VEL
LIN {X 0,Y 355.288,Z 599.445,A -85,B 0,C 180,E1 9321.197,E2 9321.197} C_VEL
LIN {X 0,Y 352.775,Z 621.65,A -85,B 0,C 180,E1 9320.521,E2 9320.521} C_VEL
LIN {X 0,Y 349.411,Z 642.885,A -85,B 0,C 180,E1 9319.627,E2 9319.627} C_VEL
LIN {X 0,Y 345.584,Z 662.737,A -85,B 0,C 180,E1 9318.531,E2 9318.531} C_VEL
LIN {X 0,Y 341.018,Z 682.531,A -85,B 0,C 180,E1 9317.135,E2 9317.135} C_VEL
LIN {X 0,Y 335.972,Z 701.696,A -85,B 0,C 180,E1 9315.456,E2 9315.456} C_VEL
LIN {X 0,Y 330.501,Z 720.54,A -85,B 0,C 180,E1 9313.441,E2 9313.441} C_VEL
LIN {X 0,Y 325.035,Z 738.024,A -85,B 0,C 180,E1 9311.167,E2 9311.167} C_VEL
LIN {X 0,Y 319.602,Z 754.233,A -85,B 0,C 180,E1 9308.615,E2 9308.615} C_VEL
LIN {X 0,Y 314.177,Z 770.121,A -85,B 0,C 180,E1 9305.616,E2 9305.616} C_VEL
LIN {X 0,Y 309.396,Z 784.17,A -85,B 0,C 180,E1 9302.44,E2 9302.44} C_VEL
LIN {X 0,Y 305.232,Z 796.772,A -85,B 0,C 180,E1 9298.997,E2 9298.997} C_VEL
LIN {X 0,Y 301.738,Z 808.178,A -85,B 0,C 180,E1 9295.225,E2 9295.225} C_VEL
LIN {X 0,Y 299.079,Z 818.289,A -85,B 0,C 180,E1 9291.133,E2 9291.133} C_VEL
LIN {X 0,Y 297.454,Z 826.124,A -85,B 0,C 180,E1 9287.203,E2 9287.203} C_VEL
LIN {X 0,Y 296.585,Z 832.168,A -85,B 0,C 180,E1 9283.25,E2 9283.25} C_VEL
LIN {X 0,Y 296.283,Z 836.839,A -85,B 0,C 180,E1 9279.124,E2 9279.124} C_VEL
LIN {X 0,Y 296.313,Z 839.53,A -85,B 0,C 180,E1 9275.474,E2 9275.474} C_VEL
LIN {X 0,Y 296.397,Z 840.884,A -85,B 0,C 180,E1 9271.738,E2 9271.738} C_VEL
LIN {X 0,Y 296.403,Z 840.869,A -85,B 0,C 180,E1 9268.452,E2 9268.452} C_VEL
LIN {X 0,Y 296.324,Z 839.62,A -85,B 0,C 180,E1 9264.771,E2 9264.771} C_VEL
LIN {X 0,Y 296.284,Z 836.859,A -85,B 0,C 180,E1 9261.068,E2 9261.068} C_VEL
LIN {X 0,Y 296.536,Z 832.561,A -85,B 0,C 180,E1 9257.14,E2 9257.14} C_VEL
LIN {X 0,Y 297.332,Z 826.573,A -85,B 0,C 180,E1 9253.188,E2 9253.188} C_VEL
LIN {X 0,Y 298.977,Z 818.504,A -85,B 0,C 180,E1 9249.031,E2 9249.031} C_VEL
LIN {X 0,Y 301.477,Z 809.037,A -85,B 0,C 180,E1 9245.088,E2 9245.088} C_VEL
LIN {X 0,Y 304.816,Z 798.138,A -85,B 0,C 180,E1 9241.384,E2 9241.384} C_VEL
LIN {X 0,Y 309.153,Z 785.227,A -85,B 0,C 180,E1 9237.746,E2 9237.746} C_VEL
LIN {X 0,Y 314.236,Z 770.873,A -85,B 0,C 180,E1 9234.387,E2 9234.387} C_VEL
LIN {X 0,Y 319.592,Z 755.912,A -85,B 0,C 180,E1 9231.458,E2 9231.458} C_VEL
LIN {X 0,Y 325.405,Z 739.27,A -85,B 0,C 180,E1 9228.768,E2 9228.768} C_VEL
LIN {X 0,Y 331.153,Z 721.981,A -85,B 0,C 180,E1 9226.44,E2 9226.44} C_VEL
LIN {X 0,Y 337.017,Z 703.269,A -85,B 0,C 180,E1 9224.355,E2 9224.355} C_VEL
LIN {X 0,Y 342.442,Z 684.149,A -85,B 0,C 180,E1 9222.624,E2 9222.624} C_VEL
LIN {X 0,Y 347.397,Z 664.248,A -85,B 0,C 180,E1 9221.179,E2 9221.179} C_VEL
LIN {X 0,Y 351.93,Z 642.995,A -85,B 0,C 180,E1 9219.962,E2 9219.962} C_VEL
LIN {X 0,Y 355.583,Z 622.213,A -85,B 0,C 180,E1 9219.06,E2 9219.06} C_VEL
LIN {X 0,Y 358.357,Z 599.971,A -85,B 0,C 180,E1 9218.368,E2 9218.368} C_VEL
LIN {X 0,Y 360.565,Z 566.718,A -85,B 0,C 180,E1 9217.631,E2 9217.631} C_VEL
LIN {X 0,Y 372.037,Z 379.475,A -85,B 0,C 180,E1 9213.743,E2 9213.743} C_VEL
LIN {X 0,Y 364.912,Z 366.255,A -85,B 0,C 180,E1 9211.373,E2 9211.373} C_VEL
LIN {X 0,Y 358.35,Z 355.353,A -85,B 0,C 180,E1 9208.909,E2 9208.909} C_VEL
LIN {X 0,Y 353.417,Z 347.777,A -85,B 0,C 180,E1 9206.779,E2 9206.779} C_VEL
LIN {X 0,Y 350.209,Z 343.051,A -85,B 0,C 180,E1 9205.222,E2 9205.222} C_VEL
LIN {X 0,Y 346.715,Z 338.013,A -85,B 0,C 180,E1 9203.272,E2 9203.272} C_VEL
LIN {X 0,Y 344.543,Z 335.082,A -85,B 0,C 180,E1 9201.896,E2 9201.896} C_VEL
LIN {X 0,Y 341.624,Z 330.839,A -85,B 0,C 180,E1 9199.67,E2 9199.67} C_VEL
LIN {X 0,Y 337.745,Z 325.58,A -85,B 0,C 180,E1 9195.278,E2 9195.278} C_VEL
LIN {X 0,Y 336.244,Z 324.331,A -85,B 0,C 180,E1 9191.095,E2 9191.095} C_VEL
LIN {X 0,Y 336.837,Z 324.882,A -85,B 0,C 180,E1 9187.335,E2 9187.335} C_VEL
LIN {X 0,Y 337.779,Z 325.931,A -85,B 0,C 180,E1 9185.437,E2 9185.437} C_VEL
LIN {X 0,Y 341.683,Z 331.314,A -85,B 0,C 180,E1 9181.091,E2 9181.091} C_VEL
LIN {X 0,Y 345.873,Z 337.387,A -85,B 0,C 180,E1 9178.013,E2 9178.013} C_VEL
LIN {X 0,Y 350.833,Z 344.477,A -85,B 0,C 180,E1 9175.22,E2 9175.22} C_VEL
LIN {X 0,Y 356.464,Z 353.299,A -85,B 0,C 180,E1 9172.588,E2 9172.588} C_VEL
LIN {X 0,Y 363.143,Z 364.378,A -85,B 0,C 180,E1 9169.932,E2 9169.932} C_VEL
LIN {X 0,Y 370.03,Z 377,A -85,B 0,C 180,E1 9167.537,E2 9167.537} C_VEL
LIN {X 0,Y 370.569,Z 378.447,A -85,B 0,C 180,E1 9167.345,E2 9167.345} C_VEL
LIN {X 0,Y 356.583,Z 575.457,A -85,B 0,C 180,E1 9163.059,E2 9163.059} C_VEL
LIN {X 0,Y 354.143,Z 596.048,A -85,B 0,C 180,E1 9162.351,E2 9162.351} C_VEL
LIN {X 0,Y 350.871,Z 616.357,A -85,B 0,C 180,E1 9161.39,E2 9161.39} C_VEL
LIN {X 0,Y 346.659,Z 637.09,A -85,B 0,C 180,E1 9160.101,E2 9160.101} C_VEL
LIN {X 0,Y 341.919,Z 656.473,A -85,B 0,C 180,E1 9158.562,E2 9158.562} C_VEL
LIN {X 0,Y 336.882,Z 674.337,A -85,B 0,C 180,E1 9156.803,E2 9156.803} C_VEL
LIN {X 0,Y 331.281,Z 691.992,A -85,B 0,C 180,E1 9154.663,E2 9154.663} C_VEL
LIN {X 0,Y 325.782,Z 707.726,A -85,B 0,C 180,E1 9152.328,E2 9152.328} C_VEL
LIN {X 0,Y 320.502,Z 721.894,A -85,B 0,C 180,E1 9149.788,E2 9149.788} C_VEL
LIN {X 0,Y 315.253,Z 735.435,A -85,B 0,C 180,E1 9146.859,E2 9146.859} C_VEL
LIN {X 0,Y 310.449,Z 747.565,A -85,B 0,C 180,E1 9143.66,E2 9143.66} C_VEL
LIN {X 0,Y 306.166,Z 758.414,A -85,B 0,C 180,E1 9140.128,E2 9140.128} C_VEL
LIN {X 0,Y 302.629,Z 767.678,A -85,B 0,C 180,E1 9136.332,E2 9136.332} C_VEL
LIN {X 0,Y 300.09,Z 774.866,A -85,B 0,C 180,E1 9132.563,E2 9132.563} C_VEL
LIN {X 0,Y 298.298,Z 780.619,A -85,B 0,C 180,E1 9128.57,E2 9128.57} C_VEL
LIN {X 0,Y 297.276,Z 784.601,A -85,B 0,C 180,E1 9124.642,E2 9124.642} C_VEL
LIN {X 0,Y 296.788,Z 786.978,A -85,B 0,C 180,E1 9120.791,E2 9120.791} C_VEL
LIN {X 0,Y 296.605,Z 787.805,A -85,B 0,C 180,E1 9117.072,E2 9117.072} C_VEL
LIN {X 0,Y 296.625,Z 787.287,A -85,B 0,C 180,E1 9113.229,E2 9113.229} C_VEL
LIN {X 0,Y 296.876,Z 785.381,A -85,B 0,C 180,E1 9109.442,E2 9109.442} C_VEL
LIN {X 0,Y 297.491,Z 781.861,A -85,B 0,C 180,E1 9105.599,E2 9105.599} C_VEL
LIN {X 0,Y 298.738,Z 776.522,A -85,B 0,C 180,E1 9101.587,E2 9101.587} C_VEL
LIN {X 0,Y 300.747,Z 769.438,A -85,B 0,C 180,E1 9097.644,E2 9097.644} C_VEL
LIN {X 0,Y 303.47,Z 760.972,A -85,B 0,C 180,E1 9093.969,E2 9093.969} C_VEL
LIN {X 0,Y 307.037,Z 750.626,A -85,B 0,C 180,E1 9090.375,E2 9090.375} C_VEL
LIN {X 0,Y 311.472,Z 738.099,A -85,B 0,C 180,E1 9086.874,E2 9086.874} C_VEL
LIN {X 0,Y 316.168,Z 724.684,A -85,B 0,C 180,E1 9083.829,E2 9083.829} C_VEL
LIN {X 0,Y 321.048,Z 710.288,A -85,B 0,C 180,E1 9081.134,E2 9081.134} C_VEL
LIN {X 0,Y 326.125,Z 694.5,A -85,B 0,C 180,E1 9078.686,E2 9078.686} C_VEL
LIN {X 0,Y 331.06,Z 677.88,A -85,B 0,C 180,E1 9076.555,E2 9076.555} C_VEL
LIN {X 0,Y 335.966,Z 659.67,A -85,B 0,C 180,E1 9074.643,E2 9074.643} C_VEL
LIN {X 0,Y 340.475,Z 640.405,A -85,B 0,C 180,E1 9073.012,E2 9073.012} C_VEL
LIN {X 0,Y 344.234,Z 621.172,A -85,B 0,C 180,E1 9071.72,E2 9071.72} C_VEL
LIN {X 0,Y 347.54,Z 600.414,A -85,B 0,C 180,E1 9070.642,E2 9070.642} C_VEL
LIN {X 0,Y 350.148,Z 578.556,A -85,B 0,C 180,E1 9069.821,E2 9069.821} C_VEL
LIN {X 0,Y 351.972,Z 553.876,A -85,B 0,C 180,E1 9069.206,E2 9069.206} C_VEL
LIN {X 0,Y 353.374,Z 529.595,A -85,B 0,C 180,E1 9068.691,E2 9068.691} C_VEL
LIN {X 0,Y 353.143,Z 522.026,A -85,B 0,C 180,E1 9068.412,E2 9068.412} C_VEL
LIN {X 0,Y 350.146,Z 502.274,A -85,B 0,C 180,E1 9067.232,E2 9067.232} C_VEL
LIN {X 0,Y 350.037,Z 495.768,A -85,B 0,C 180,E1 9066.999,E2 9066.999} C_VEL
LIN {X 0,Y 357.234,Z 377.006,A -85,B 0,C 180,E1 9064.469,E2 9064.469} C_VEL
LIN {X 0,Y 348.21,Z 361.407,A -85,B 0,C 180,E1 9061.997,E2 9061.997} C_VEL
LIN {X 0,Y 337.882,Z 345.206,A -85,B 0,C 180,E1 9058.901,E2 9058.901} C_VEL
LIN {X 0,Y 329.047,Z 332.526,A -85,B 0,C 180,E1 9055.971,E2 9055.971} C_VEL
LIN {X 0,Y 319.78,Z 319.823,A -85,B 0,C 180,E1 9052.501,E2 9052.501} C_VEL
LIN {X 0,Y 314.604,Z 313.307,A -85,B 0,C 180,E1 9050.342,E2 9050.342} C_VEL
LIN {X 0,Y 309.943,Z 307.496,A -85,B 0,C 180,E1 9048.242,E2 9048.242} C_VEL
LIN {X 0,Y 306.277,Z 303.065,A -85,B 0,C 180,E1 9046.443,E2 9046.443} C_VEL
LIN {X 0,Y 303.655,Z 299.378,A -85,B 0,C 180,E1 9044.798,E2 9044.798} C_VEL
LIN {X 0,Y 302.772,Z 297.817,A -85,B 0,C 180,E1 9043.904,E2 9043.904} C_VEL
LIN {X 0,Y 300.635,Z 294.028,A -85,B 0,C 180,E1 9041.56,E2 9041.56} C_VEL
LIN {X 0,Y 300.009,Z 292.837,A -85,B 0,C 180,E1 9040.782,E2 9040.782} C_VEL
LIN {X 0,Y 297.593,Z 289.001,A -85,B 0,C 180,E1 9037.86,E2 9037.86} C_VEL
LIN {X 0,Y 296.836,Z 287.488,A -85,B 0,C 180,E1 9036.714,E2 9036.714} C_VEL
LIN {X 0,Y 294.303,Z 283.686,A -85,B 0,C 180,E1 9032.925,E2 9032.925} C_VEL
LIN {X 0,Y 293.46,Z 281.951,A -85,B 0,C 180,E1 9031.188,E2 9031.188} C_VEL
LIN {X 0,Y 290.419,Z 277.047,A -85,B 0,C 180,E1 9022.679,E2 9022.679} C_VEL
LIN {X 0,Y 290.347,Z 276.57,A -85,B 0,C 180,E1 9018.677,E2 9018.677} C_VEL
LIN {X 0,Y 290.347,Z 276.555,A -85,B 0,C 180,E1 9013.947,E2 9013.947} C_VEL
LIN {X 0,Y 290.422,Z 277.021,A -85,B 0,C 180,E1 9009.71,E2 9009.71} C_VEL
LIN {X 0,Y 293.957,Z 282.508,A -85,B 0,C 180,E1 9000.527,E2 9000.527} C_VEL
LIN {X 0,Y 296.646,Z 287.281,A -85,B 0,C 180,E1 8996.059,E2 8996.059} C_VEL
LIN {X 0,Y 297.706,Z 288.61,A -85,B 0,C 180,E1 8994.796,E2 8994.796} C_VEL
LIN {X 0,Y 299.937,Z 292.674,A -85,B 0,C 180,E1 8991.899,E2 8991.899} C_VEL
LIN {X 0,Y 300.996,Z 294.135,A -85,B 0,C 180,E1 8990.824,E2 8990.824} C_VEL
LIN {X 0,Y 303.289,Z 298.15,A -85,B 0,C 180,E1 8988.397,E2 8988.397} C_VEL
LIN {X 0,Y 304.089,Z 299.326,A -85,B 0,C 180,E1 8987.658,E2 8987.658} C_VEL
LIN {X 0,Y 306.001,Z 302.583,A -85,B 0,C 180,E1 8986.199,E2 8986.199} C_VEL
LIN {X 0,Y 308.666,Z 305.54,A -85,B 0,C 180,E1 8984.883,E2 8984.883} C_VEL
LIN {X 0,Y 313.335,Z 311.292,A -85,B 0,C 180,E1 8982.687,E2 8982.687} C_VEL
LIN {X 0,Y 317.799,Z 316.882,A -85,B 0,C 180,E1 8980.756,E2 8980.756} C_VEL
LIN {X 0,Y 323.291,Z 323.983,A -85,B 0,C 180,E1 8978.572,E2 8978.572} C_VEL
LIN {X 0,Y 332.302,Z 335.982,A -85,B 0,C 180,E1 8975.328,E2 8975.328} C_VEL
LIN {X 0,Y 342.213,Z 350.366,A -85,B 0,C 180,E1 8972.128,E2 8972.128} C_VEL
LIN {X 0,Y 351.475,Z 364.639,A -85,B 0,C 180,E1 8969.435,E2 8969.435} C_VEL
LIN {X 0,Y 361.352,Z 381.129,A -85,B 0,C 180,E1 8966.802,E2 8966.802} C_VEL
LIN {X 0,Y 362.045,Z 382.679,A -85,B 0,C 180,E1 8966.614,E2 8966.614} C_VEL
LIN {X 0,Y 349.792,Z 599.114,A -85,B 0,C 180,E1 8962.149,E2 8962.149} C_VEL
LIN {X 0,Y 347.202,Z 621.345,A -85,B 0,C 180,E1 8961.469,E2 8961.469} C_VEL
LIN {X 0,Y 343.845,Z 641.996,A -85,B 0,C 180,E1 8960.599,E2 8960.599} C_VEL
LIN {X 0,Y 339.892,Z 661.956,A -85,B 0,C 180,E1 8959.498,E2 8959.498} C_VEL
LIN {X 0,Y 335.148,Z 681.877,A -85,B 0,C 180,E1 8958.086,E2 8958.086} C_VEL
LIN {X 0,Y 329.943,Z 700.978,A -85,B 0,C 180,E1 8956.404,E2 8956.404} C_VEL
LIN {X 0,Y 324.351,Z 719.571,A -85,B 0,C 180,E1 8954.404,E2 8954.404} C_VEL
LIN {X 0,Y 318.573,Z 737.355,A -85,B 0,C 180,E1 8952.07,E2 8952.07} C_VEL
LIN {X 0,Y 312.914,Z 753.609,A -85,B 0,C 180,E1 8949.481,E2 8949.481} C_VEL
LIN {X 0,Y 307.387,Z 769.067,A -85,B 0,C 180,E1 8946.528,E2 8946.528} C_VEL
LIN {X 0,Y 302.35,Z 783.186,A -85,B 0,C 180,E1 8943.293,E2 8943.293} C_VEL
LIN {X 0,Y 297.93,Z 795.82,A -85,B 0,C 180,E1 8939.779,E2 8939.779} C_VEL
LIN {X 0,Y 294.272,Z 807.094,A -85,B 0,C 180,E1 8935.993,E2 8935.993} C_VEL
LIN {X 0,Y 291.489,Z 816.969,A -85,B 0,C 180,E1 8931.953,E2 8931.953} C_VEL
LIN {X 0,Y 289.669,Z 824.943,A -85,B 0,C 180,E1 8927.888,E2 8927.888} C_VEL
LIN {X 0,Y 288.672,Z 831.121,A -85,B 0,C 180,E1 8923.825,E2 8923.825} C_VEL
LIN {X 0,Y 288.315,Z 835.749,A -85,B 0,C 180,E1 8919.781,E2 8919.781} C_VEL
LIN {X 0,Y 288.322,Z 838.591,A -85,B 0,C 180,E1 8915.969,E2 8915.969} C_VEL
LIN {X 0,Y 288.417,Z 840.122,A -85,B 0,C 180,E1 8912.183,E2 8912.183} C_VEL
LIN {X 0,Y 288.436,Z 840.184,A -85,B 0,C 180,E1 8908.607,E2 8908.607} C_VEL
LIN {X 0,Y 288.358,Z 839.085,A -85,B 0,C 180,E1 8905.025,E2 8905.025} C_VEL
LIN {X 0,Y 288.3,Z 836.324,A -85,B 0,C 180,E1 8901.019,E2 8901.019} C_VEL
LIN {X 0,Y 288.557,Z 832.112,A -85,B 0,C 180,E1 8896.982,E2 8896.982} C_VEL
LIN {X 0,Y 289.459,Z 825.849,A -85,B 0,C 180,E1 8892.717,E2 8892.717} C_VEL
LIN {X 0,Y 291.25,Z 817.79,A -85,B 0,C 180,E1 8888.447,E2 8888.447} C_VEL
LIN {X 0,Y 294.006,Z 808.091,A -85,B 0,C 180,E1 8884.32,E2 8884.32} C_VEL
LIN {X 0,Y 297.725,Z 796.826,A -85,B 0,C 180,E1 8880.416,E2 8880.416} C_VEL
LIN {X 0,Y 302.215,Z 784.259,A -85,B 0,C 180,E1 8876.83,E2 8876.83} C_VEL
LIN {X 0,Y 307.801,Z 769.314,A -85,B 0,C 180,E1 8873.292,E2 8873.292} C_VEL
LIN {X 0,Y 313.638,Z 753.873,A -85,B 0,C 180,E1 8870.267,E2 8870.267} C_VEL
LIN {X 0,Y 319.844,Z 736.914,A -85,B 0,C 180,E1 8867.526,E2 8867.526} C_VEL
LIN {X 0,Y 325.81,Z 719.66,A -85,B 0,C 180,E1 8865.225,E2 8865.225} C_VEL
LIN {X 0,Y 331.982,Z 700.559,A -85,B 0,C 180,E1 8863.133,E2 8863.133} C_VEL
LIN {X 0,Y 337.51,Z 681.789,A -85,B 0,C 180,E1 8861.451,E2 8861.451} C_VEL
LIN {X 0,Y 342.384,Z 662.679,A -85,B 0,C 180,E1 8860.081,E2 8860.081} C_VEL
LIN {X 0,Y 347.069,Z 641.232,A -85,B 0,C 180,E1 8858.87,E2 8858.87} C_VEL
LIN {X 0,Y 350.793,Z 620.325,A -85,B 0,C 180,E1 8857.981,E2 8857.981} C_VEL
LIN {X 0,Y 353.664,Z 597.756,A -85,B 0,C 180,E1 8857.288,E2 8857.288} C_VEL
LIN {X 0,Y 356.906,Z 547.851,A -85,B 0,C 180,E1 8856.212,E2 8856.212} C_VEL
LIN {X 0,Y 367.516,Z 383.334,A -85,B 0,C 180,E1 8852.756,E2 8852.756} C_VEL
LIN {X 0,Y 360.903,Z 370.918,A -85,B 0,C 180,E1 8850.418,E2 8850.418} C_VEL
LIN {X 0,Y 354.518,Z 360.046,A -85,B 0,C 180,E1 8847.825,E2 8847.825} C_VEL
LIN {X 0,Y 349.031,Z 351.478,A -85,B 0,C 180,E1 8845.223,E2 8845.223} C_VEL
LIN {X 0,Y 344.878,Z 345.395,A -85,B 0,C 180,E1 8842.862,E2 8842.862} C_VEL
LIN {X 0,Y 342.813,Z 342.518,A -85,B 0,C 180,E1 8841.481,E2 8841.481} C_VEL
LIN {X 0,Y 339.997,Z 338.381,A -85,B 0,C 180,E1 8839.232,E2 8839.232} C_VEL
LIN {X 0,Y 336.554,Z 333.434,A -85,B 0,C 180,E1 8835.082,E2 8835.082} C_VEL
LIN {X 0,Y 335.165,Z 332.254,A -85,B 0,C 180,E1 8831.008,E2 8831.008} C_VEL
LIN {X 0,Y 335.818,Z 332.87,A -85,B 0,C 180,E1 8827.185,E2 8827.185} C_VEL
LIN {X 0,Y 336.624,Z 333.901,A -85,B 0,C 180,E1 8825.541,E2 8825.541} C_VEL
LIN {X 0,Y 340.236,Z 339.082,A -85,B 0,C 180,E1 8821.348,E2 8821.348} C_VEL
LIN {X 0,Y 344.199,Z 344.976,A -85,B 0,C 180,E1 8818.337,E2 8818.337} C_VEL
LIN {X 0,Y 348.776,Z 351.797,A -85,B 0,C 180,E1 8815.645,E2 8815.645} C_VEL
LIN {X 0,Y 354.066,Z 360.34,A -85,B 0,C 180,E1 8813.068,E2 8813.068} C_VEL
LIN {X 0,Y 360.361,Z 371.114,A -85,B 0,C 180,E1 8810.459,E2 8810.459} C_VEL
LIN {X 0,Y 366.142,Z 382.118,A -85,B 0,C 180,E1 8808.335,E2 8808.335} C_VEL
LIN {X 0,Y 351.775,Z 576.098,A -85,B 0,C 180,E1 8804.087,E2 8804.087} C_VEL
LIN {X 0,Y 349.227,Z 596.813,A -85,B 0,C 180,E1 8803.372,E2 8803.372} C_VEL
LIN {X 0,Y 345.869,Z 616.882,A -85,B 0,C 180,E1 8802.417,E2 8802.417} C_VEL
LIN {X 0,Y 341.622,Z 637.021,A -85,B 0,C 180,E1 8801.164,E2 8801.164} C_VEL
LIN {X 0,Y 336.884,Z 655.792,A -85,B 0,C 180,E1 8799.683,E2 8799.683} C_VEL
LIN {X 0,Y 331.43,Z 674.504,A -85,B 0,C 180,E1 8797.847,E2 8797.847} C_VEL
LIN {X 0,Y 325.713,Z 691.757,A -85,B 0,C 180,E1 8795.747,E2 8795.747} C_VEL
LIN {X 0,Y 319.893,Z 707.726,A -85,B 0,C 180,E1 8793.373,E2 8793.373} C_VEL
LIN {X 0,Y 314.012,Z 722.84,A -85,B 0,C 180,E1 8790.638,E2 8790.638} C_VEL
LIN {X 0,Y 308.516,Z 736.267,A -85,B 0,C 180,E1 8787.676,E2 8787.676} C_VEL
LIN {X 0,Y 303.515,Z 748.236,A -85,B 0,C 180,E1 8784.46,E2 8784.46} C_VEL
LIN {X 0,Y 298.892,Z 759.275,A -85,B 0,C 180,E1 8780.787,E2 8780.787} C_VEL
LIN {X 0,Y 295.224,Z 768.245,A -85,B 0,C 180,E1 8777.018,E2 8777.018} C_VEL
LIN {X 0,Y 292.471,Z 775.501,A -85,B 0,C 180,E1 8773.138,E2 8773.138} C_VEL
LIN {X 0,Y 290.479,Z 781.405,A -85,B 0,C 180,E1 8768.934,E2 8768.934} C_VEL
LIN {X 0,Y 289.344,Z 785.453,A -85,B 0,C 180,E1 8764.765,E2 8764.765} C_VEL
LIN {X 0,Y 288.829,Z 787.775,A -85,B 0,C 180,E1 8760.822,E2 8760.822} C_VEL
LIN {X 0,Y 288.637,Z 788.537,A -85,B 0,C 180,E1 8756.989,E2 8756.989} C_VEL
LIN {X 0,Y 288.669,Z 787.891,A -85,B 0,C 180,E1 8752.884,E2 8752.884} C_VEL
